LIN {X 0,Y 573.25,Z 574.073,A -85,B 0,C 180,E1 -2307.355,E2 -2307.355} C_VEL
LIN {X 0,Y 573.251,Z 574.074,A -85,B 0,C 180,E1 -2309.824,E2 -2309.824} C_VEL
LIN {X 0,Y 573.282,Z 574.075,A -85,B 0,C 180,E1 -2312.235,E2 -2312.235} C_VEL
LIN {X 0,Y 573.263,Z 574.072,A -85,B 0,C 180,E1 -2315.12,E2 -2315.12} C_VEL
LIN {X 0,Y 573.23,Z 574.076,A -85,B 0,C 180,E1 -2317.662,E2 -2317.662} C_VEL
LIN {X 0,Y 573.27,Z 574.075,A -85,B 0,C 180,E1 -2320.728,E2 -2320.728} C_VEL
LIN {X 0,Y 573.245,Z 574.074,A -85,B 0,C 180,E1 -2323.621,E2 -2323.621} C_VEL
LIN {X 0,Y 573.265,Z 574.072,A -85,B 0,C 180,E1 -2325.807,E2 -2325.807} C_VEL
LIN {X 0,Y 573.254,Z 574.076,A -85,B 0,C 180,E1 -2328.745,E2 -2328.745} C_VEL
LIN {X 0,Y 573.3,Z 574.067,A -85,B 0,C 180,E1 -2331.541,E2 -2331.541} C_VEL
LIN {X 0,Y 573.283,Z 574.078,A -85,B 0,C 180,E1 -2334.372,E2 -2334.372} C_VEL
LIN {X 0,Y 573.301,Z 574.07,A -85,B 0,C 180,E1 -2337.892,E2 -2337.892} C_VEL
LIN {X 0,Y 573.328,Z 574.067,A -85,B 0,C 180,E1 -2340.702,E2 -2340.702} C_VEL
LIN {X 0,Y 573.232,Z 574.076,A -85,B 0,C 180,E1 -2343.514,E2 -2343.514} C_VEL
LIN {X 0,Y 573.292,Z 574.069,A -85,B 0,C 180,E1 -2345.628,E2 -2345.628} C_VEL
LIN {X 0,Y 573.301,Z 574.074,A -85,B 0,C 180,E1 -2348.459,E2 -2348.459} C_VEL
LIN {X 0,Y 573.291,Z 574.068,A -85,B 0,C 180,E1 -2351.312,E2 -2351.312} C_VEL
LIN {X 0,Y 573.273,Z 574.08,A -85,B 0,C 180,E1 -2354.425,E2 -2354.425} C_VEL
LIN {X 0,Y 573.304,Z 574.233,A -85,B 0,C 180,E1 -2357.432,E2 -2357.432} C_VEL
LIN {X 0,Y 573.275,Z 587.865,A -85,B 0,C 180,E1 -2360.076,E2 -2360.076} C_VEL
LIN {X 0,Y 573.251,Z 593.888,A -85,B 0,C 180,E1 -2361.233,E2 -2361.233} C_VEL
LIN {X 0,Y 574.072,Z 600.547,A -85,B 0,C 180,E1 -2361.34,E2 -2361.34} C_VEL
LIN {X 0,Y 574.064,Z 601.305,A -85,B 0,C 180,E1 -2361.349,E2 -2361.349} C_VEL
LIN {X 0,Y 573.377,Z 607.149,A -85,B 0,C 180,E1 -2361.406,E2 -2361.406} C_VEL
LIN {X 0,Y 567.79,Z 626.154,A -85,B 0,C 180,E1 -2361.512,E2 -2361.512} C_VEL
LIN {X 0,Y 567.122,Z 631.997,A -85,B 0,C 180,E1 -2361.57,E2 -2361.57} C_VEL
LIN {X 0,Y 566.935,Z 700.341,A -85,B 0,C 180,E1 -2362.455,E2 -2362.455} C_VEL
LIN {X 0,Y 566.844,Z 713.428,A -85,B 0,C 180,E1 -2362.772,E2 -2362.772} C_VEL
LIN {X 0,Y 566.759,Z 725.192,A -85,B 0,C 180,E1 -2363.185,E2 -2363.185} C_VEL
LIN {X 0,Y 566.603,Z 736.809,A -85,B 0,C 180,E1 -2363.735,E2 -2363.735} C_VEL
LIN {X 0,Y 566.457,Z 748.669,A -85,B 0,C 180,E1 -2364.461,E2 -2364.461} C_VEL
LIN {X 0,Y 566.329,Z 758.973,A -85,B 0,C 180,E1 -2365.256,E2 -2365.256} C_VEL
LIN {X 0,Y 566.211,Z 768.35,A -85,B 0,C 180,E1 -2366.145,E2 -2366.145} C_VEL
LIN {X 0,Y 566.092,Z 777.03,A -85,B 0,C 180,E1 -2367.154,E2 -2367.154} C_VEL
LIN {X 0,Y 566.019,Z 785.144,A -85,B 0,C 180,E1 -2368.335,E2 -2368.335} C_VEL
LIN {X 0,Y 565.978,Z 790.458,A -85,B 0,C 180,E1 -2369.298,E2 -2369.298} C_VEL
LIN {X 0,Y 565.921,Z 796.115,A -85,B 0,C 180,E1 -2370.608,E2 -2370.608} C_VEL
LIN {X 0,Y 565.867,Z 799.979,A -85,B 0,C 180,E1 -2371.86,E2 -2371.86} C_VEL
LIN {X 0,Y 565.839,Z 802.539,A -85,B 0,C 180,E1 -2373.127,E2 -2373.127} C_VEL
LIN {X 0,Y 565.858,Z 803.553,A -85,B 0,C 180,E1 -2373.98,E2 -2373.98} C_VEL
LIN {X 0,Y 565.846,Z 803.984,A -85,B 0,C 180,E1 -2374.943,E2 -2374.943} C_VEL
LIN {X 0,Y 565.821,Z 803.511,A -85,B 0,C 180,E1 -2376.163,E2 -2376.163} C_VEL
LIN {X 0,Y 565.843,Z 801.631,A -85,B 0,C 180,E1 -2377.488,E2 -2377.488} C_VEL
LIN {X 0,Y 565.868,Z 799.217,A -85,B 0,C 180,E1 -2378.516,E2 -2378.516} C_VEL
LIN {X 0,Y 565.92,Z 795.465,A -85,B 0,C 180,E1 -2379.651,E2 -2379.651} C_VEL
LIN {X 0,Y 565.941,Z 789.748,A -85,B 0,C 180,E1 -2380.933,E2 -2380.933} C_VEL
LIN {X 0,Y 566.008,Z 782.933,A -85,B 0,C 180,E1 -2382.106,E2 -2382.106} C_VEL
LIN {X 0,Y 566.108,Z 776.028,A -85,B 0,C 180,E1 -2383.063,E2 -2383.063} C_VEL
LIN {X 0,Y 566.186,Z 767.481,A -85,B 0,C 180,E1 -2384.037,E2 -2384.037} C_VEL
LIN {X 0,Y 566.366,Z 757.173,A -85,B 0,C 180,E1 -2384.985,E2 -2384.985} C_VEL
LIN {X 0,Y 566.477,Z 746.803,A -85,B 0,C 180,E1 -2385.755,E2 -2385.755} C_VEL
LIN {X 0,Y 566.635,Z 735.245,A -85,B 0,C 180,E1 -2386.437,E2 -2386.437} C_VEL
LIN {X 0,Y 566.756,Z 722.817,A -85,B 0,C 180,E1 -2387,E2 -2387} C_VEL
LIN {X 0,Y 566.89,Z 709.938,A -85,B 0,C 180,E1 -2387.421,E2 -2387.421} C_VEL
LIN {X 0,Y 566.982,Z 696.718,A -85,B 0,C 180,E1 -2387.693,E2 -2387.693} C_VEL
LIN {X 0,Y 567.083,Z 599.04,A -85,B 0,C 180,E1 -2388.942,E2 -2388.942} C_VEL
LIN {X 0,Y 566.197,Z 593.841,A -85,B 0,C 180,E1 -2389.042,E2 -2389.042} C_VEL
LIN {X 0,Y 566.362,Z 579.311,A -85,B 0,C 180,E1 -2391.879,E2 -2391.879} C_VEL
LIN {X 0,Y 566.259,Z 574.948,A -85,B 0,C 180,E1 -2392.788,E2 -2392.788} C_VEL
LIN {X 0,Y 566.22,Z 574.957,A -85,B 0,C 180,E1 -2396.046,E2 -2396.046} C_VEL
LIN {X 0,Y 566.191,Z 574.953,A -85,B 0,C 180,E1 -2398.579,E2 -2398.579} C_VEL
LIN {X 0,Y 566.191,Z 574.951,A -85,B 0,C 180,E1 -2401.048,E2 -2401.048} C_VEL
LIN {X 0,Y 566.214,Z 574.95,A -85,B 0,C 180,E1 -2403.46,E2 -2403.46} C_VEL
LIN {X 0,Y 566.198,Z 574.956,A -85,B 0,C 180,E1 -2405.82,E2 -2405.82} C_VEL
LIN {X 0,Y 566.208,Z 574.95,A -85,B 0,C 180,E1 -2408.903,E2 -2408.903} C_VEL
LIN {X 0,Y 566.208,Z 574.949,A -85,B 0,C 180,E1 -2411.173,E2 -2411.173} C_VEL
LIN {X 0,Y 566.217,Z 574.948,A -85,B 0,C 180,E1 -2413.413,E2 -2413.413} C_VEL
LIN {X 0,Y 566.201,Z 574.96,A -85,B 0,C 180,E1 -2416.36,E2 -2416.36} C_VEL
LIN {X 0,Y 566.235,Z 574.951,A -85,B 0,C 180,E1 -2418.676,E2 -2418.676} C_VEL
LIN {X 0,Y 566.23,Z 574.947,A -85,B 0,C 180,E1 -2421.435,E2 -2421.435} C_VEL
LIN {X 0,Y 566.26,Z 574.951,A -85,B 0,C 180,E1 -2424.303,E2 -2424.303} C_VEL
LIN {X 0,Y 566.284,Z 574.941,A -85,B 0,C 180,E1 -2427.867,E2 -2427.867} C_VEL
LIN {X 0,Y 566.304,Z 574.945,A -85,B 0,C 180,E1 -2430.712,E2 -2430.712} C_VEL
LIN {X 0,Y 566.278,Z 574.947,A -85,B 0,C 180,E1 -2432.846,E2 -2432.846} C_VEL
LIN {X 0,Y 566.26,Z 574.943,A -85,B 0,C 180,E1 -2435.699,E2 -2435.699} C_VEL
LIN {X 0,Y 566.237,Z 574.954,A -85,B 0,C 180,E1 -2438.566,E2 -2438.566} C_VEL
LIN {X 0,Y 566.246,Z 574.945,A -85,B 0,C 180,E1 -2441.455,E2 -2441.455} C_VEL
LIN {X 0,Y 566.238,Z 574.951,A -85,B 0,C 180,E1 -2444.507,E2 -2444.507} C_VEL
LIN {X 0,Y 566.204,Z 574.953,A -85,B 0,C 180,E1 -2447.332,E2 -2447.332} C_VEL
LIN {X 0,Y 566.212,Z 574.951,A -85,B 0,C 180,E1 -2450.338,E2 -2450.338} C_VEL
LIN {X 0,Y 566.173,Z 574.959,A -85,B 0,C 180,E1 -2453.281,E2 -2453.281} C_VEL
LIN {X 0,Y 566.218,Z 574.949,A -85,B 0,C 180,E1 -2455.749,E2 -2455.749} C_VEL
LIN {X 0,Y 566.207,Z 574.95,A -85,B 0,C 180,E1 -2458.203,E2 -2458.203} C_VEL
LIN {X 0,Y 566.195,Z 574.961,A -85,B 0,C 180,E1 -2461.077,E2 -2461.077} C_VEL
LIN {X 0,Y 566.216,Z 574.95,A -85,B 0,C 180,E1 -2463.735,E2 -2463.735} C_VEL
LIN {X 0,Y 566.204,Z 574.951,A -85,B 0,C 180,E1 -2466.57,E2 -2466.57} C_VEL
LIN {X 0,Y 566.226,Z 574.951,A -85,B 0,C 180,E1 -2469.687,E2 -2469.687} C_VEL
LIN {X 0,Y 566.205,Z 574.953,A -85,B 0,C 180,E1 -2472.918,E2 -2472.918} C_VEL
LIN {X 0,Y 566.202,Z 574.951,A -85,B 0,C 180,E1 -2476.049,E2 -2476.049} C_VEL
LIN {X 0,Y 566.184,Z 574.954,A -85,B 0,C 180,E1 -2478.861,E2 -2478.861} C_VEL
LIN {X 0,Y 566.192,Z 574.959,A -85,B 0,C 180,E1 -2481.637,E2 -2481.637} C_VEL
LIN {X 0,Y 566.167,Z 574.955,A -85,B 0,C 180,E1 -2484.308,E2 -2484.308} C_VEL
LIN {X 0,Y 566.225,Z 574.948,A -85,B 0,C 180,E1 -2486.898,E2 -2486.898} C_VEL
LIN {X 0,Y 566.185,Z 574.959,A -85,B 0,C 180,E1 -2489.408,E2 -2489.408} C_VEL
LIN {X 0,Y 566.216,Z 574.956,A -85,B 0,C 180,E1 -2491.858,E2 -2491.858} C_VEL
LIN {X 0,Y 566.218,Z 574.95,A -85,B 0,C 180,E1 -2494.251,E2 -2494.251} C_VEL
LIN {X 0,Y 566.174,Z 574.953,A -85,B 0,C 180,E1 -2496.719,E2 -2496.719} C_VEL
LIN {X 0,Y 566.213,Z 574.956,A -85,B 0,C 180,E1 -2499.663,E2 -2499.663} C_VEL
LIN {X 0,Y 566.204,Z 574.95,A -85,B 0,C 180,E1 -2502.669,E2 -2502.669} C_VEL
LIN {X 0,Y 566.239,Z 574.951,A -85,B 0,C 180,E1 -2505.627,E2 -2505.627} C_VEL
LIN {X 0,Y 566.24,Z 574.946,A -85,B 0,C 180,E1 -2508.675,E2 -2508.675} C_VEL
LIN {X 0,Y 566.232,Z 574.948,A -85,B 0,C 180,E1 -2511.434,E2 -2511.434} C_VEL
LIN {X 0,Y 566.261,Z 574.949,A -85,B 0,C 180,E1 -2514.302,E2 -2514.302} C_VEL
LIN {X 0,Y 566.286,Z 574.945,A -85,B 0,C 180,E1 -2517.866,E2 -2517.866} C_VEL
LIN {X 0,Y 566.306,Z 574.94,A -85,B 0,C 180,E1 -2520.711,E2 -2520.711} C_VEL
LIN {X 0,Y 566.278,Z 574.942,A -85,B 0,C 180,E1 -2522.846,E2 -2522.846} C_VEL
LIN {X 0,Y 566.258,Z 574.945,A -85,B 0,C 180,E1 -2525.698,E2 -2525.698} C_VEL
LIN {X 0,Y 566.233,Z 574.953,A -85,B 0,C 180,E1 -2528.566,E2 -2528.566} C_VEL
LIN {X 0,Y 566.247,Z 574.944,A -85,B 0,C 180,E1 -2531.454,E2 -2531.454} C_VEL
LIN {X 0,Y 566.24,Z 574.955,A -85,B 0,C 180,E1 -2534.506,E2 -2534.506} C_VEL
LIN {X 0,Y 566.204,Z 574.95,A -85,B 0,C 180,E1 -2537.332,E2 -2537.332} C_VEL
LIN {X 0,Y 566.214,Z 574.955,A -85,B 0,C 180,E1 -2540.337,E2 -2540.337} C_VEL
LIN {X 0,Y 566.175,Z 574.955,A -85,B 0,C 180,E1 -2543.281,E2 -2543.281} C_VEL
LIN {X 0,Y 566.215,Z 574.948,A -85,B 0,C 180,E1 -2545.749,E2 -2545.749} C_VEL
LIN {X 0,Y 566.208,Z 574.952,A -85,B 0,C 180,E1 -2548.202,E2 -2548.202} C_VEL
LIN {X 0,Y 566.195,Z 574.956,A -85,B 0,C 180,E1 -2551.076,E2 -2551.076} C_VEL
LIN {X 0,Y 566.218,Z 574.948,A -85,B 0,C 180,E1 -2553.734,E2 -2553.734} C_VEL
LIN {X 0,Y 566.205,Z 574.955,A -85,B 0,C 180,E1 -2556.57,E2 -2556.57} C_VEL
LIN {X 0,Y 566.221,Z 574.948,A -85,B 0,C 180,E1 -2559.686,E2 -2559.686} C_VEL
LIN {X 0,Y 566.217,Z 574.948,A -85,B 0,C 180,E1 -2562.087,E2 -2562.087} C_VEL
LIN {X 0,Y 566.174,Z 574.964,A -85,B 0,C 180,E1 -2565.036,E2 -2565.036} C_VEL
LIN {X 0,Y 566.194,Z 574.951,A -85,B 0,C 180,E1 -2567.91,E2 -2567.91} C_VEL
LIN {X 0,Y 566.225,Z 574.951,A -85,B 0,C 180,E1 -2570.727,E2 -2570.727} C_VEL
LIN {X 0,Y 566.19,Z 574.953,A -85,B 0,C 180,E1 -2573.788,E2 -2573.788} C_VEL
LIN {X 0,Y 566.218,Z 574.949,A -85,B 0,C 180,E1 -2576.265,E2 -2576.265} C_VEL
LIN {X 0,Y 566.193,Z 574.956,A -85,B 0,C 180,E1 -2578.924,E2 -2578.924} C_VEL
LIN {X 0,Y 566.217,Z 574.952,A -85,B 0,C 180,E1 -2581.857,E2 -2581.857} C_VEL
LIN {X 0,Y 566.215,Z 574.952,A -85,B 0,C 180,E1 -2584.25,E2 -2584.25} C_VEL
LIN {X 0,Y 566.26,Z 575.009,A -85,B 0,C 180,E1 -2585.431,E2 -2585.431} C_VEL
LIN {X 0,Y 567.273,Z 580.215,A -85,B 0,C 180,E1 -2586.22,E2 -2586.22} C_VEL
LIN {X 0,Y 567.133,Z 596.227,A -85,B 0,C 180,E1 -2588.47,E2 -2588.47} C_VEL
LIN {X 0,Y 566.794,Z 618.681,A -85,B 0,C 180,E1 -2591.567,E2 -2591.567} C_VEL
LIN {X 0,Y 566.549,Z 637.787,A -85,B 0,C 180,E1 -2594.162,E2 -2594.162} C_VEL
LIN {X 0,Y 566.428,Z 651.349,A -85,B 0,C 180,E1 -2595.986,E2 -2595.986} C_VEL
LIN {X 0,Y 567.183,Z 658.149,A -85,B 0,C 180,E1 -2596.094,E2 -2596.094} C_VEL
LIN {X 0,Y 566.989,Z 759.91,A -85,B 0,C 180,E1 -2597.403,E2 -2597.403} C_VEL
LIN {X 0,Y 566.841,Z 772.433,A -85,B 0,C 180,E1 -2597.695,E2 -2597.695} C_VEL
LIN {X 0,Y 566.764,Z 785.356,A -85,B 0,C 180,E1 -2598.148,E2 -2598.148} C_VEL
LIN {X 0,Y 566.629,Z 797.14,A -85,B 0,C 180,E1 -2598.707,E2 -2598.707} C_VEL
LIN {X 0,Y 566.449,Z 809.192,A -85,B 0,C 180,E1 -2599.454,E2 -2599.454} C_VEL
LIN {X 0,Y 566.319,Z 819.592,A -85,B 0,C 180,E1 -2600.265,E2 -2600.265} C_VEL
LIN {X 0,Y 566.207,Z 828.105,A -85,B 0,C 180,E1 -2601.073,E2 -2601.073} C_VEL
LIN {X 0,Y 566.113,Z 835.955,A -85,B 0,C 180,E1 -2601.971,E2 -2601.971} C_VEL
LIN {X 0,Y 566.004,Z 843.617,A -85,B 0,C 180,E1 -2603.046,E2 -2603.046} C_VEL
LIN {X 0,Y 566.004,Z 850.676,A -85,B 0,C 180,E1 -2604.298,E2 -2604.298} C_VEL
LIN {X 0,Y 565.934,Z 855.369,A -85,B 0,C 180,E1 -2605.369,E2 -2605.369} C_VEL
LIN {X 0,Y 565.927,Z 858.955,A -85,B 0,C 180,E1 -2606.439,E2 -2606.439} C_VEL
LIN {X 0,Y 565.878,Z 860.806,A -85,B 0,C 180,E1 -2607.152,E2 -2607.152} C_VEL
LIN {X 0,Y 565.846,Z 863.185,A -85,B 0,C 180,E1 -2608.576,E2 -2608.576} C_VEL
LIN {X 0,Y 565.839,Z 864,A -85,B 0,C 180,E1 -2609.999,E2 -2609.999} C_VEL
LIN {X 0,Y 565.846,Z 863.187,A -85,B 0,C 180,E1 -2611.423,E2 -2611.423} C_VEL
LIN {X 0,Y 565.878,Z 860.812,A -85,B 0,C 180,E1 -2612.847,E2 -2612.847} C_VEL
LIN {X 0,Y 565.926,Z 857.898,A -85,B 0,C 180,E1 -2613.916,E2 -2613.916} C_VEL
LIN {X 0,Y 565.878,Z 853.952,A -85,B 0,C 180,E1 -2614.987,E2 -2614.987} C_VEL
LIN {X 0,Y 566.001,Z 848.871,A -85,B 0,C 180,E1 -2616.058,E2 -2616.058} C_VEL
LIN {X 0,Y 566.04,Z 842.474,A -85,B 0,C 180,E1 -2617.131,E2 -2617.131} C_VEL
LIN {X 0,Y 566.133,Z 834.485,A -85,B 0,C 180,E1 -2618.207,E2 -2618.207} C_VEL
LIN {X 0,Y 566.228,Z 826.344,A -85,B 0,C 180,E1 -2619.105,E2 -2619.105} C_VEL
LIN {X 0,Y 566.342,Z 816.411,A -85,B 0,C 180,E1 -2620.004,E2 -2620.004} C_VEL
LIN {X 0,Y 566.524,Z 805.296,A -85,B 0,C 180,E1 -2620.807,E2 -2620.807} C_VEL
LIN {X 0,Y 566.659,Z 794.194,A -85,B 0,C 180,E1 -2621.445,E2 -2621.445} C_VEL
LIN {X 0,Y 566.75,Z 782.006,A -85,B 0,C 180,E1 -2621.987,E2 -2621.987} C_VEL
LIN {X 0,Y 566.887,Z 769.211,A -85,B 0,C 180,E1 -2622.393,E2 -2622.393} C_VEL
LIN {X 0,Y 566.981,Z 757.164,A -85,B 0,C 180,E1 -2622.641,E2 -2622.641} C_VEL
LIN {X 0,Y 567.032,Z 655.343,A -85,B 0,C 180,E1 -2623.945,E2 -2623.945} C_VEL
LIN {X 0,Y 566.444,Z 651.276,A -85,B 0,C 180,E1 -2624.023,E2 -2624.023} C_VEL
LIN {X 0,Y 566.692,Z 627.248,A -85,B 0,C 180,E1 -2627.265,E2 -2627.265} C_VEL
LIN {X 0,Y 566.952,Z 606.411,A -85,B 0,C 180,E1 -2630.119,E2 -2630.119} C_VEL
LIN {X 0,Y 567.307,Z 584.574,A -85,B 0,C 180,E1 -2633.161,E2 -2633.161} C_VEL
LIN {X 0,Y 567.077,Z 578.976,A -85,B 0,C 180,E1 -2633.965,E2 -2633.965} C_VEL
LIN {X 0,Y 566.233,Z 574.957,A -85,B 0,C 180,E1 -2634.593,E2 -2634.593} C_VEL
LIN {X 0,Y 566.211,Z 574.952,A -85,B 0,C 180,E1 -2637.338,E2 -2637.338} C_VEL
LIN {X 0,Y 566.2,Z 574.953,A -85,B 0,C 180,E1 -2639.768,E2 -2639.768} C_VEL
LIN {X 0,Y 566.203,Z 574.96,A -85,B 0,C 180,E1 -2642.429,E2 -2642.429} C_VEL
LIN {X 0,Y 566.211,Z 574.953,A -85,B 0,C 180,E1 -2644.993,E2 -2644.993} C_VEL
LIN {X 0,Y 566.193,Z 574.952,A -85,B 0,C 180,E1 -2647.46,E2 -2647.46} C_VEL
LIN {X 0,Y 566.224,Z 574.954,A -85,B 0,C 180,E1 -2650.196,E2 -2650.196} C_VEL
LIN {X 0,Y 566.197,Z 574.954,A -85,B 0,C 180,E1 -2653.053,E2 -2653.053} C_VEL
LIN {X 0,Y 566.198,Z 574.955,A -85,B 0,C 180,E1 -2656.047,E2 -2656.047} C_VEL
LIN {X 0,Y 566.208,Z 574.954,A -85,B 0,C 180,E1 -2658.863,E2 -2658.863} C_VEL
LIN {X 0,Y 566.187,Z 574.953,A -85,B 0,C 180,E1 -2661.637,E2 -2661.637} C_VEL
LIN {X 0,Y 566.207,Z 574.957,A -85,B 0,C 180,E1 -2664.311,E2 -2664.311} C_VEL
LIN {X 0,Y 566.223,Z 574.951,A -85,B 0,C 180,E1 -2666.898,E2 -2666.898} C_VEL
LIN {X 0,Y 566.188,Z 574.952,A -85,B 0,C 180,E1 -2669.407,E2 -2669.407} C_VEL
LIN {X 0,Y 566.222,Z 574.949,A -85,B 0,C 180,E1 -2671.858,E2 -2671.858} C_VEL
LIN {X 0,Y 566.221,Z 574.955,A -85,B 0,C 180,E1 -2674.251,E2 -2674.251} C_VEL
LIN {X 0,Y 566.185,Z 574.958,A -85,B 0,C 180,E1 -2676.713,E2 -2676.713} C_VEL
LIN {X 0,Y 566.207,Z 574.95,A -85,B 0,C 180,E1 -2679.662,E2 -2679.662} C_VEL
LIN {X 0,Y 566.196,Z 574.957,A -85,B 0,C 180,E1 -2682.668,E2 -2682.668} C_VEL
LIN {X 0,Y 566.226,Z 574.948,A -85,B 0,C 180,E1 -2685.626,E2 -2685.626} C_VEL
LIN {X 0,Y 566.226,Z 574.953,A -85,B 0,C 180,E1 -2688.675,E2 -2688.675} C_VEL
LIN {X 0,Y 566.241,Z 574.946,A -85,B 0,C 180,E1 -2691.434,E2 -2691.434} C_VEL
LIN {X 0,Y 566.252,Z 574.955,A -85,B 0,C 180,E1 -2694.302,E2 -2694.302} C_VEL
LIN {X 0,Y 566.272,Z 574.945,A -85,B 0,C 180,E1 -2697.866,E2 -2697.866} C_VEL
LIN {X 0,Y 566.298,Z 574.943,A -85,B 0,C 180,E1 -2700.711,E2 -2700.711} C_VEL
LIN {X 0,Y 566.272,Z 574.945,A -85,B 0,C 180,E1 -2702.845,E2 -2702.845} C_VEL
LIN {X 0,Y 566.26,Z 574.946,A -85,B 0,C 180,E1 -2705.698,E2 -2705.698} C_VEL
LIN {X 0,Y 566.242,Z 574.952,A -85,B 0,C 180,E1 -2708.565,E2 -2708.565} C_VEL
LIN {X 0,Y 566.243,Z 574.946,A -85,B 0,C 180,E1 -2711.454,E2 -2711.454} C_VEL
LIN {X 0,Y 566.226,Z 574.957,A -85,B 0,C 180,E1 -2714.507,E2 -2714.507} C_VEL
LIN {X 0,Y 566.271,Z 575.092,A -85,B 0,C 180,E1 -2717.376,E2 -2717.376} C_VEL
LIN {X 0,Y 566.241,Z 588.233,A -85,B 0,C 180,E1 -2719.957,E2 -2719.957} C_VEL
LIN {X 0,Y 566.19,Z 593.854,A -85,B 0,C 180,E1 -2721.051,E2 -2721.051} C_VEL
LIN {X 0,Y 567.187,Z 600.576,A -85,B 0,C 180,E1 -2721.17,E2 -2721.17} C_VEL
LIN {X 0,Y 567.122,Z 631.997,A -85,B 0,C 180,E1 -2721.57,E2 -2721.57} C_VEL
LIN {X 0,Y 566.416,Z 635.921,A -85,B 0,C 180,E1 -2721.603,E2 -2721.603} C_VEL
LIN {X 0,Y 560.748,Z 648.204,A -85,B 0,C 180,E1 -2721.623,E2 -2721.623} C_VEL
LIN {X 0,Y 560.188,Z 652.117,A -85,B 0,C 180,E1 -2721.66,E2 -2721.66} C_VEL
LIN {X 0,Y 560.024,Z 700.973,A -85,B 0,C 180,E1 -2722.31,E2 -2722.31} C_VEL
LIN {X 0,Y 559.912,Z 713.82,A -85,B 0,C 180,E1 -2722.631,E2 -2722.631} C_VEL
LIN {X 0,Y 559.798,Z 725.266,A -85,B 0,C 180,E1 -2723.039,E2 -2723.039} C_VEL
LIN {X 0,Y 559.612,Z 737.425,A -85,B 0,C 180,E1 -2723.626,E2 -2723.626} C_VEL
LIN {X 0,Y 559.457,Z 748.173,A -85,B 0,C 180,E1 -2724.293,E2 -2724.293} C_VEL
LIN {X 0,Y 559.327,Z 758.049,A -85,B 0,C 180,E1 -2725.052,E2 -2725.052} C_VEL
LIN {X 0,Y 559.187,Z 767.063,A -85,B 0,C 180,E1 -2725.896,E2 -2725.896} C_VEL
LIN {X 0,Y 559.023,Z 775.909,A -85,B 0,C 180,E1 -2726.91,E2 -2726.91} C_VEL
LIN {X 0,Y 558.964,Z 783.819,A -85,B 0,C 180,E1 -2728.033,E2 -2728.033} C_VEL
LIN {X 0,Y 558.896,Z 790.145,A -85,B 0,C 180,E1 -2729.161,E2 -2729.161} C_VEL
LIN {X 0,Y 558.827,Z 794.778,A -85,B 0,C 180,E1 -2730.202,E2 -2730.202} C_VEL
LIN {X 0,Y 558.827,Z 798.325,A -85,B 0,C 180,E1 -2731.221,E2 -2731.221} C_VEL
LIN {X 0,Y 558.758,Z 801.643,A -85,B 0,C 180,E1 -2732.574,E2 -2732.574} C_VEL
LIN {X 0,Y 558.764,Z 803.491,A -85,B 0,C 180,E1 -2733.89,E2 -2733.89} C_VEL
LIN {X 0,Y 558.752,Z 803.981,A -85,B 0,C 180,E1 -2735.159,E2 -2735.159} C_VEL
LIN {X 0,Y 558.732,Z 803.288,A -85,B 0,C 180,E1 -2736.389,E2 -2736.389} C_VEL
LIN {X 0,Y 558.755,Z 801.489,A -85,B 0,C 180,E1 -2737.59,E2 -2737.59} C_VEL
LIN {X 0,Y 558.807,Z 798.043,A -85,B 0,C 180,E1 -2738.964,E2 -2738.964} C_VEL
LIN {X 0,Y 558.854,Z 792.793,A -85,B 0,C 180,E1 -2740.364,E2 -2740.364} C_VEL
LIN {X 0,Y 558.896,Z 786.646,A -85,B 0,C 180,E1 -2741.586,E2 -2741.586} C_VEL
LIN {X 0,Y 558.981,Z 779.074,A -85,B 0,C 180,E1 -2742.76,E2 -2742.76} C_VEL
LIN {X 0,Y 559.12,Z 770.156,A -85,B 0,C 180,E1 -2743.864,E2 -2743.864} C_VEL
LIN {X 0,Y 559.301,Z 760.04,A -85,B 0,C 180,E1 -2744.864,E2 -2744.864} C_VEL
LIN {X 0,Y 559.452,Z 749.138,A -85,B 0,C 180,E1 -2745.729,E2 -2745.729} C_VEL
LIN {X 0,Y 559.629,Z 738.117,A -85,B 0,C 180,E1 -2746.424,E2 -2746.424} C_VEL
LIN {X 0,Y 559.79,Z 727.068,A -85,B 0,C 180,E1 -2746.974,E2 -2746.974} C_VEL
LIN {X 0,Y 559.918,Z 714.065,A -85,B 0,C 180,E1 -2747.456,E2 -2747.456} C_VEL
LIN {X 0,Y 559.992,Z 701.471,A -85,B 0,C 180,E1 -2747.771,E2 -2747.771} C_VEL
LIN {X 0,Y 560.115,Z 670.961,A -85,B 0,C 180,E1 -2748.189,E2 -2748.189} C_VEL
LIN {X 0,Y 560.13,Z 599.387,A -85,B 0,C 180,E1 -2749.113,E2 -2749.113} C_VEL
LIN {X 0,Y 559.168,Z 593.853,A -85,B 0,C 180,E1 -2749.219,E2 -2749.219} C_VEL
LIN {X 0,Y 559.363,Z 578.134,A -85,B 0,C 180,E1 -2752.331,E2 -2752.331} C_VEL
LIN {X 0,Y 559.233,Z 575.824,A -85,B 0,C 180,E1 -2752.8,E2 -2752.8} C_VEL
LIN {X 0,Y 559.176,Z 575.834,A -85,B 0,C 180,E1 -2756.05,E2 -2756.05} C_VEL
LIN {X 0,Y 559.153,Z 575.828,A -85,B 0,C 180,E1 -2758.982,E2 -2758.982} C_VEL
LIN {X 0,Y 559.168,Z 575.83,A -85,B 0,C 180,E1 -2761.619,E2 -2761.619} C_VEL
LIN {X 0,Y 559.179,Z 575.832,A -85,B 0,C 180,E1 -2763.904,E2 -2763.904} C_VEL
LIN {X 0,Y 559.155,Z 575.831,A -85,B 0,C 180,E1 -2766.568,E2 -2766.568} C_VEL
LIN {X 0,Y 559.179,Z 575.825,A -85,B 0,C 180,E1 -2769.396,E2 -2769.396} C_VEL
LIN {X 0,Y 559.152,Z 575.831,A -85,B 0,C 180,E1 -2771.687,E2 -2771.687} C_VEL
LIN {X 0,Y 559.169,Z 575.831,A -85,B 0,C 180,E1 -2773.949,E2 -2773.949} C_VEL
LIN {X 0,Y 559.175,Z 575.834,A -85,B 0,C 180,E1 -2776.185,E2 -2776.185} C_VEL
LIN {X 0,Y 559.206,Z 575.827,A -85,B 0,C 180,E1 -2778.605,E2 -2778.605} C_VEL
LIN {X 0,Y 559.188,Z 575.824,A -85,B 0,C 180,E1 -2781.326,E2 -2781.326} C_VEL
LIN {X 0,Y 559.229,Z 575.825,A -85,B 0,C 180,E1 -2784.231,E2 -2784.231} C_VEL
LIN {X 0,Y 559.255,Z 575.817,A -85,B 0,C 180,E1 -2787.84,E2 -2787.84} C_VEL
LIN {X 0,Y 559.274,Z 575.821,A -85,B 0,C 180,E1 -2790.721,E2 -2790.721} C_VEL
LIN {X 0,Y 559.244,Z 575.822,A -85,B 0,C 180,E1 -2792.882,E2 -2792.882} C_VEL
LIN {X 0,Y 559.23,Z 575.819,A -85,B 0,C 180,E1 -2795.771,E2 -2795.771} C_VEL
LIN {X 0,Y 559.195,Z 575.833,A -85,B 0,C 180,E1 -2798.675,E2 -2798.675} C_VEL
LIN {X 0,Y 559.209,Z 575.821,A -85,B 0,C 180,E1 -2801.601,E2 -2801.601} C_VEL
LIN {X 0,Y 559.204,Z 575.828,A -85,B 0,C 180,E1 -2804.596,E2 -2804.596} C_VEL
LIN {X 0,Y 559.163,Z 575.828,A -85,B 0,C 180,E1 -2807.557,E2 -2807.557} C_VEL
LIN {X 0,Y 559.17,Z 575.826,A -85,B 0,C 180,E1 -2809.838,E2 -2809.838} C_VEL
LIN {X 0,Y 559.145,Z 575.83,A -85,B 0,C 180,E1 -2812.153,E2 -2812.153} C_VEL
LIN {X 0,Y 559.18,Z 575.83,A -85,B 0,C 180,E1 -2815.299,E2 -2815.299} C_VEL
LIN {X 0,Y 559.185,Z 575.825,A -85,B 0,C 180,E1 -2817.713,E2 -2817.713} C_VEL
LIN {X 0,Y 559.157,Z 575.828,A -85,B 0,C 180,E1 -2820.183,E2 -2820.183} C_VEL
LIN {X 0,Y 559.161,Z 575.831,A -85,B 0,C 180,E1 -2822.716,E2 -2822.716} C_VEL
LIN {X 0,Y 559.14,Z 575.838,A -85,B 0,C 180,E1 -2825.324,E2 -2825.324} C_VEL
LIN {X 0,Y 559.138,Z 575.83,A -85,B 0,C 180,E1 -2828.018,E2 -2828.018} C_VEL
LIN {X 0,Y 559.159,Z 575.83,A -85,B 0,C 180,E1 -2830.813,E2 -2830.813} C_VEL
LIN {X 0,Y 559.142,Z 575.833,A -85,B 0,C 180,E1 -2833.735,E2 -2833.735} C_VEL
LIN {X 0,Y 559.151,Z 575.83,A -85,B 0,C 180,E1 -2836.804,E2 -2836.804} C_VEL
LIN {X 0,Y 559.162,Z 575.833,A -85,B 0,C 180,E1 -2839.188,E2 -2839.188} C_VEL
LIN {X 0,Y 559.138,Z 575.833,A -85,B 0,C 180,E1 -2841.983,E2 -2841.983} C_VEL
LIN {X 0,Y 559.136,Z 575.831,A -85,B 0,C 180,E1 -2844.787,E2 -2844.787} C_VEL
LIN {X 0,Y 559.161,Z 575.834,A -85,B 0,C 180,E1 -2847.365,E2 -2847.365} C_VEL
LIN {X 0,Y 559.153,Z 575.831,A -85,B 0,C 180,E1 -2850.143,E2 -2850.143} C_VEL
LIN {X 0,Y 559.174,Z 575.827,A -85,B 0,C 180,E1 -2853.098,E2 -2853.098} C_VEL
LIN {X 0,Y 559.16,Z 575.833,A -85,B 0,C 180,E1 -2855.495,E2 -2855.495} C_VEL
LIN {X 0,Y 559.177,Z 575.825,A -85,B 0,C 180,E1 -2858.624,E2 -2858.624} C_VEL
LIN {X 0,Y 559.166,Z 575.826,A -85,B 0,C 180,E1 -2860.926,E2 -2860.926} C_VEL
LIN {X 0,Y 559.17,Z 575.836,A -85,B 0,C 180,E1 -2863.948,E2 -2863.948} C_VEL
LIN {X 0,Y 559.175,Z 575.832,A -85,B 0,C 180,E1 -2866.184,E2 -2866.184} C_VEL
LIN {X 0,Y 559.199,Z 575.823,A -85,B 0,C 180,E1 -2869.134,E2 -2869.134} C_VEL
LIN {X 0,Y 559.205,Z 575.832,A -85,B 0,C 180,E1 -2872.054,E2 -2872.054} C_VEL
LIN {X 0,Y 559.259,Z 575.815,A -85,B 0,C 180,E1 -2874.953,E2 -2874.953} C_VEL
LIN {X 0,Y 559.258,Z 575.82,A -85,B 0,C 180,E1 -2877.84,E2 -2877.84} C_VEL
LIN {X 0,Y 559.277,Z 575.815,A -85,B 0,C 180,E1 -2880.72,E2 -2880.72} C_VEL
LIN {X 0,Y 559.244,Z 575.818,A -85,B 0,C 180,E1 -2882.881,E2 -2882.881} C_VEL
LIN {X 0,Y 559.228,Z 575.821,A -85,B 0,C 180,E1 -2885.77,E2 -2885.77} C_VEL
LIN {X 0,Y 559.192,Z 575.828,A -85,B 0,C 180,E1 -2888.674,E2 -2888.674} C_VEL
LIN {X 0,Y 559.211,Z 575.821,A -85,B 0,C 180,E1 -2891.6,E2 -2891.6} C_VEL
LIN {X 0,Y 559.206,Z 575.83,A -85,B 0,C 180,E1 -2894.596,E2 -2894.596} C_VEL
LIN {X 0,Y 559.148,Z 575.829,A -85,B 0,C 180,E1 -2897.557,E2 -2897.557} C_VEL
LIN {X 0,Y 559.172,Z 575.827,A -85,B 0,C 180,E1 -2899.838,E2 -2899.838} C_VEL
LIN {X 0,Y 559.146,Z 575.832,A -85,B 0,C 180,E1 -2902.153,E2 -2902.153} C_VEL
LIN {X 0,Y 559.181,Z 575.826,A -85,B 0,C 180,E1 -2905.298,E2 -2905.298} C_VEL
LIN {X 0,Y 559.153,Z 575.828,A -85,B 0,C 180,E1 -2907.714,E2 -2907.714} C_VEL
LIN {X 0,Y 559.158,Z 575.83,A -85,B 0,C 180,E1 -2910.183,E2 -2910.183} C_VEL
LIN {X 0,Y 559.162,Z 575.836,A -85,B 0,C 180,E1 -2912.715,E2 -2912.715} C_VEL
LIN {X 0,Y 559.134,Z 575.833,A -85,B 0,C 180,E1 -2915.324,E2 -2915.324} C_VEL
LIN {X 0,Y 559.139,Z 575.83,A -85,B 0,C 180,E1 -2918.017,E2 -2918.017} C_VEL
LIN {X 0,Y 559.163,Z 575.835,A -85,B 0,C 180,E1 -2920.812,E2 -2920.812} C_VEL
LIN {X 0,Y 559.153,Z 575.835,A -85,B 0,C 180,E1 -2923.196,E2 -2923.196} C_VEL
LIN {X 0,Y 559.143,Z 575.83,A -85,B 0,C 180,E1 -2926.266,E2 -2926.266} C_VEL
LIN {X 0,Y 559.161,Z 575.836,A -85,B 0,C 180,E1 -2929.187,E2 -2929.187} C_VEL
LIN {X 0,Y 559.138,Z 575.83,A -85,B 0,C 180,E1 -2931.982,E2 -2931.982} C_VEL
LIN {X 0,Y 559.14,Z 575.834,A -85,B 0,C 180,E1 -2934.786,E2 -2934.786} C_VEL
LIN {X 0,Y 559.179,Z 575.834,A -85,B 0,C 180,E1 -2937.361,E2 -2937.361} C_VEL
LIN {X 0,Y 559.15,Z 575.83,A -85,B 0,C 180,E1 -2940.143,E2 -2940.143} C_VEL
LIN {X 0,Y 559.174,Z 575.834,A -85,B 0,C 180,E1 -2943.097,E2 -2943.097} C_VEL
LIN {X 0,Y 559.211,Z 575.841,A -85,B 0,C 180,E1 -2945.251,E2 -2945.251} C_VEL
LIN {X 0,Y 560.456,Z 583.194,A -85,B 0,C 180,E1 -2946.342,E2 -2946.342} C_VEL
LIN {X 0,Y 560.088,Z 603.669,A -85,B 0,C 180,E1 -2949.238,E2 -2949.238} C_VEL
LIN {X 0,Y 559.758,Z 625.505,A -85,B 0,C 180,E1 -2952.273,E2 -2952.273} C_VEL
LIN {X 0,Y 559.463,Z 646.221,A -85,B 0,C 180,E1 -2955.11,E2 -2955.11} C_VEL
LIN {X 0,Y 559.439,Z 651.349,A -85,B 0,C 180,E1 -2955.808,E2 -2955.808} C_VEL
LIN {X 0,Y 560.294,Z 658.175,A -85,B 0,C 180,E1 -2955.92,E2 -2955.92} C_VEL
LIN {X 0,Y 560.084,Z 759.91,A -85,B 0,C 180,E1 -2957.245,E2 -2957.245} C_VEL
LIN {X 0,Y 559.923,Z 772.433,A -85,B 0,C 180,E1 -2957.541,E2 -2957.541} C_VEL
LIN {X 0,Y 559.792,Z 785.358,A -85,B 0,C 180,E1 -2957.998,E2 -2957.998} C_VEL
LIN {X 0,Y 559.67,Z 796.795,A -85,B 0,C 180,E1 -2958.546,E2 -2958.546} C_VEL
LIN {X 0,Y 559.511,Z 807.899,A -85,B 0,C 180,E1 -2959.231,E2 -2959.231} C_VEL
LIN {X 0,Y 559.311,Z 818.532,A -85,B 0,C 180,E1 -2960.05,E2 -2960.05} C_VEL
LIN {X 0,Y 559.162,Z 828.106,A -85,B 0,C 180,E1 -2960.96,E2 -2960.96} C_VEL
LIN {X 0,Y 559.05,Z 835.955,A -85,B 0,C 180,E1 -2961.869,E2 -2961.869} C_VEL
LIN {X 0,Y 558.945,Z 843.617,A -85,B 0,C 180,E1 -2962.958,E2 -2962.958} C_VEL
LIN {X 0,Y 558.935,Z 850.676,A -85,B 0,C 180,E1 -2964.226,E2 -2964.226} C_VEL
LIN {X 0,Y 558.827,Z 855.369,A -85,B 0,C 180,E1 -2965.31,E2 -2965.31} C_VEL
LIN {X 0,Y 558.837,Z 858.955,A -85,B 0,C 180,E1 -2966.394,E2 -2966.394} C_VEL
LIN {X 0,Y 558.8,Z 860.806,A -85,B 0,C 180,E1 -2967.116,E2 -2967.116} C_VEL
LIN {X 0,Y 558.745,Z 863.184,A -85,B 0,C 180,E1 -2968.558,E2 -2968.558} C_VEL
LIN {X 0,Y 558.74,Z 864,A -85,B 0,C 180,E1 -2969.999,E2 -2969.999} C_VEL
LIN {X 0,Y 558.745,Z 863.187,A -85,B 0,C 180,E1 -2971.441,E2 -2971.441} C_VEL
LIN {X 0,Y 558.799,Z 860.812,A -85,B 0,C 180,E1 -2972.883,E2 -2972.883} C_VEL
LIN {X 0,Y 558.844,Z 857.898,A -85,B 0,C 180,E1 -2973.965,E2 -2973.965} C_VEL
LIN {X 0,Y 558.798,Z 853.952,A -85,B 0,C 180,E1 -2975.05,E2 -2975.05} C_VEL
LIN {X 0,Y 558.921,Z 848.871,A -85,B 0,C 180,E1 -2976.135,E2 -2976.135} C_VEL
LIN {X 0,Y 558.977,Z 842.474,A -85,B 0,C 180,E1 -2977.222,E2 -2977.222} C_VEL
LIN {X 0,Y 559.098,Z 834.485,A -85,B 0,C 180,E1 -2978.311,E2 -2978.311} C_VEL
LIN {X 0,Y 559.183,Z 826.344,A -85,B 0,C 180,E1 -2979.22,E2 -2979.22} C_VEL
LIN {X 0,Y 559.355,Z 816.411,A -85,B 0,C 180,E1 -2980.13,E2 -2980.13} C_VEL
LIN {X 0,Y 559.529,Z 805.376,A -85,B 0,C 180,E1 -2980.939,E2 -2980.939} C_VEL
LIN {X 0,Y 559.702,Z 793.16,A -85,B 0,C 180,E1 -2981.643,E2 -2981.643} C_VEL
LIN {X 0,Y 559.83,Z 780.792,A -85,B 0,C 180,E1 -2982.184,E2 -2982.184} C_VEL
LIN {X 0,Y 559.934,Z 767.382,A -85,B 0,C 180,E1 -2982.596,E2 -2982.596} C_VEL
LIN {X 0,Y 560.087,Z 754.146,A -85,B 0,C 180,E1 -2982.845,E2 -2982.845} C_VEL
LIN {X 0,Y 560.12,Z 655.762,A -85,B 0,C 180,E1 -2984.116,E2 -2984.116} C_VEL
LIN {X 0,Y 559.457,Z 651.276,A -85,B 0,C 180,E1 -2984.202,E2 -2984.202} C_VEL
LIN {X 0,Y 559.71,Z 628.861,A -85,B 0,C 180,E1 -2987.265,E2 -2987.265} C_VEL
LIN {X 0,Y 560.023,Z 607.775,A -85,B 0,C 180,E1 -2990.188,E2 -2990.188} C_VEL
LIN {X 0,Y 560.428,Z 585.939,A -85,B 0,C 180,E1 -2993.266,E2 -2993.266} C_VEL
LIN {X 0,Y 560.437,Z 581.953,A -85,B 0,C 180,E1 -2993.834,E2 -2993.834} C_VEL
LIN {X 0,Y 559.205,Z 575.832,A -85,B 0,C 180,E1 -2994.747,E2 -2994.747} C_VEL
LIN {X 0,Y 559.188,Z 575.827,A -85,B 0,C 180,E1 -2997.711,E2 -2997.711} C_VEL
LIN {X 0,Y 559.152,Z 575.834,A -85,B 0,C 180,E1 -3000.182,E2 -3000.182} C_VEL
LIN {X 0,Y 559.173,Z 575.835,A -85,B 0,C 180,E1 -3002.713,E2 -3002.713} C_VEL
LIN {X 0,Y 559.156,Z 575.83,A -85,B 0,C 180,E1 -3005.321,E2 -3005.321} C_VEL
LIN {X 0,Y 559.132,Z 575.835,A -85,B 0,C 180,E1 -3008.016,E2 -3008.016} C_VEL
LIN {X 0,Y 559.173,Z 575.833,A -85,B 0,C 180,E1 -3010.81,E2 -3010.81} C_VEL
LIN {X 0,Y 559.137,Z 575.833,A -85,B 0,C 180,E1 -3013.733,E2 -3013.733} C_VEL
LIN {X 0,Y 559.164,Z 575.833,A -85,B 0,C 180,E1 -3016.8,E2 -3016.8} C_VEL
LIN {X 0,Y 559.172,Z 575.828,A -85,B 0,C 180,E1 -3019.189,E2 -3019.189} C_VEL
LIN {X 0,Y 559.131,Z 575.834,A -85,B 0,C 180,E1 -3021.982,E2 -3021.982} C_VEL
LIN {X 0,Y 559.154,Z 575.833,A -85,B 0,C 180,E1 -3024.782,E2 -3024.782} C_VEL
LIN {X 0,Y 559.168,Z 575.827,A -85,B 0,C 180,E1 -3027.361,E2 -3027.361} C_VEL
LIN {X 0,Y 559.183,Z 575.83,A -85,B 0,C 180,E1 -3030.134,E2 -3030.134} C_VEL
LIN {X 0,Y 559.176,Z 575.826,A -85,B 0,C 180,E1 -3033.169,E2 -3033.169} C_VEL
LIN {X 0,Y 559.15,Z 575.829,A -85,B 0,C 180,E1 -3035.494,E2 -3035.494} C_VEL
LIN {X 0,Y 559.164,Z 575.833,A -85,B 0,C 180,E1 -3038.623,E2 -3038.623} C_VEL
LIN {X 0,Y 559.164,Z 575.83,A -85,B 0,C 180,E1 -3040.926,E2 -3040.926} C_VEL
LIN {X 0,Y 559.161,Z 575.831,A -85,B 0,C 180,E1 -3043.948,E2 -3043.948} C_VEL
LIN {X 0,Y 559.166,Z 575.834,A -85,B 0,C 180,E1 -3046.184,E2 -3046.184} C_VEL
LIN {X 0,Y 559.188,Z 575.825,A -85,B 0,C 180,E1 -3049.133,E2 -3049.133} C_VEL
LIN {X 0,Y 559.201,Z 575.828,A -85,B 0,C 180,E1 -3052.053,E2 -3052.053} C_VEL
LIN {X 0,Y 559.252,Z 575.818,A -85,B 0,C 180,E1 -3054.953,E2 -3054.953} C_VEL
LIN {X 0,Y 559.244,Z 575.821,A -85,B 0,C 180,E1 -3057.839,E2 -3057.839} C_VEL
LIN {X 0,Y 559.268,Z 575.819,A -85,B 0,C 180,E1 -3060.72,E2 -3060.72} C_VEL
LIN {X 0,Y 559.237,Z 575.821,A -85,B 0,C 180,E1 -3062.881,E2 -3062.881} C_VEL
LIN {X 0,Y 559.23,Z 575.823,A -85,B 0,C 180,E1 -3065.77,E2 -3065.77} C_VEL
LIN {X 0,Y 559.197,Z 575.828,A -85,B 0,C 180,E1 -3068.674,E2 -3068.674} C_VEL
LIN {X 0,Y 559.201,Z 575.825,A -85,B 0,C 180,E1 -3071.6,E2 -3071.6} C_VEL
LIN {X 0,Y 559.191,Z 575.832,A -85,B 0,C 180,E1 -3074.596,E2 -3074.596} C_VEL
LIN {X 0,Y 559.252,Z 575.917,A -85,B 0,C 180,E1 -3077.312,E2 -3077.312} C_VEL
LIN {X 0,Y 559.237,Z 587.012,A -85,B 0,C 180,E1 -3079.522,E2 -3079.522} C_VEL
LIN {X 0,Y 559.176,Z 593.843,A -85,B 0,C 180,E1 -3080.869,E2 -3080.869} C_VEL
LIN {X 0,Y 560.297,Z 600.391,A -85,B 0,C 180,E1 -3080.994,E2 -3080.994} C_VEL
LIN {X 0,Y 560.188,Z 652.117,A -85,B 0,C 180,E1 -3081.66,E2 -3081.66} C_VEL
LIN {X 0,Y 559.685,Z 657.956,A -85,B 0,C 180,E1 -3081.723,E2 -3081.723} C_VEL
LIN {X 0,Y 556.856,Z 667.442,A -85,B 0,C 180,E1 -3081.777,E2 -3081.777} C_VEL
LIN {X 0,Y 553.886,Z 676.93,A -85,B 0,C 180,E1 -3081.829,E2 -3081.829} C_VEL
LIN {X 0,Y 553.171,Z 682.783,A -85,B 0,C 180,E1 -3081.888,E2 -3081.888} C_VEL
LIN {X 0,Y 553.108,Z 702.341,A -85,B 0,C 180,E1 -3082.176,E2 -3082.176} C_VEL
LIN {X 0,Y 552.961,Z 714.256,A -85,B 0,C 180,E1 -3082.488,E2 -3082.488} C_VEL
LIN {X 0,Y 552.831,Z 725.927,A -85,B 0,C 180,E1 -3082.913,E2 -3082.913} C_VEL
LIN {X 0,Y 552.63,Z 737.79,A -85,B 0,C 180,E1 -3083.501,E2 -3083.501} C_VEL
LIN {X 0,Y 552.467,Z 749.099,A -85,B 0,C 180,E1 -3084.221,E2 -3084.221} C_VEL
LIN {X 0,Y 552.288,Z 758.85,A -85,B 0,C 180,E1 -3084.993,E2 -3084.993} C_VEL
LIN {X 0,Y 552.133,Z 767.708,A -85,B 0,C 180,E1 -3085.846,E2 -3085.846} C_VEL
LIN {X 0,Y 551.987,Z 777.185,A -85,B 0,C 180,E1 -3086.971,E2 -3086.971} C_VEL
LIN {X 0,Y 551.889,Z 784.839,A -85,B 0,C 180,E1 -3088.111,E2 -3088.111} C_VEL
LIN {X 0,Y 551.805,Z 791.475,A -85,B 0,C 180,E1 -3089.364,E2 -3089.364} C_VEL
LIN {X 0,Y 551.734,Z 796.587,A -85,B 0,C 180,E1 -3090.632,E2 -3090.632} C_VEL
LIN {X 0,Y 551.675,Z 800.313,A -85,B 0,C 180,E1 -3091.917,E2 -3091.917} C_VEL
LIN {X 0,Y 551.659,Z 802.745,A -85,B 0,C 180,E1 -3093.217,E2 -3093.217} C_VEL
LIN {X 0,Y 551.655,Z 803.646,A -85,B 0,C 180,E1 -3094.099,E2 -3094.099} C_VEL
LIN {X 0,Y 551.666,Z 803.934,A -85,B 0,C 180,E1 -3095.382,E2 -3095.382} C_VEL
LIN {X 0,Y 551.645,Z 802.876,A -85,B 0,C 180,E1 -3096.783,E2 -3096.783} C_VEL
LIN {X 0,Y 551.658,Z 801.041,A -85,B 0,C 180,E1 -3097.829,E2 -3097.829} C_VEL
LIN {X 0,Y 551.712,Z 798.057,A -85,B 0,C 180,E1 -3099.01,E2 -3099.01} C_VEL
LIN {X 0,Y 551.741,Z 793.955,A -85,B 0,C 180,E1 -3100.159,E2 -3100.159} C_VEL
LIN {X 0,Y 551.813,Z 787.722,A -85,B 0,C 180,E1 -3101.474,E2 -3101.474} C_VEL
LIN {X 0,Y 551.914,Z 780.245,A -85,B 0,C 180,E1 -3102.694,E2 -3102.694} C_VEL
LIN {X 0,Y 552.071,Z 771.661,A -85,B 0,C 180,E1 -3103.805,E2 -3103.805} C_VEL
LIN {X 0,Y 552.225,Z 762.941,A -85,B 0,C 180,E1 -3104.723,E2 -3104.723} C_VEL
LIN {X 0,Y 552.408,Z 752.765,A -85,B 0,C 180,E1 -3105.596,E2 -3105.596} C_VEL
LIN {X 0,Y 552.559,Z 741.894,A -85,B 0,C 180,E1 -3106.347,E2 -3106.347} C_VEL
LIN {X 0,Y 552.794,Z 730.515,A -85,B 0,C 180,E1 -3106.968,E2 -3106.968} C_VEL
LIN {X 0,Y 552.954,Z 717.768,A -85,B 0,C 180,E1 -3107.491,E2 -3107.491} C_VEL
LIN {X 0,Y 553.058,Z 704.466,A -85,B 0,C 180,E1 -3107.872,E2 -3107.872} C_VEL
LIN {X 0,Y 553.17,Z 689.133,A -85,B 0,C 180,E1 -3108.119,E2 -3108.119} C_VEL
LIN {X 0,Y 553.352,Z 600.793,A -85,B 0,C 180,E1 -3109.271,E2 -3109.271} C_VEL
LIN {X 0,Y 552.155,Z 593.845,A -85,B 0,C 180,E1 -3109.404,E2 -3109.404} C_VEL
LIN {X 0,Y 552.316,Z 578.001,A -85,B 0,C 180,E1 -3112.585,E2 -3112.585} C_VEL
LIN {X 0,Y 552.195,Z 576.701,A -85,B 0,C 180,E1 -3112.862,E2 -3112.862} C_VEL
LIN {X 0,Y 552.138,Z 576.712,A -85,B 0,C 180,E1 -3115.941,E2 -3115.941} C_VEL
LIN {X 0,Y 552.115,Z 576.707,A -85,B 0,C 180,E1 -3118.541,E2 -3118.541} C_VEL
LIN {X 0,Y 552.123,Z 576.706,A -85,B 0,C 180,E1 -3121.438,E2 -3121.438} C_VEL
LIN {X 0,Y 552.128,Z 576.709,A -85,B 0,C 180,E1 -3124.357,E2 -3124.357} C_VEL
LIN {X 0,Y 552.109,Z 576.707,A -85,B 0,C 180,E1 -3126.759,E2 -3126.759} C_VEL
LIN {X 0,Y 552.12,Z 576.704,A -85,B 0,C 180,E1 -3129.121,E2 -3129.121} C_VEL
LIN {X 0,Y 552.128,Z 576.704,A -85,B 0,C 180,E1 -3131.445,E2 -3131.445} C_VEL
LIN {X 0,Y 552.118,Z 576.707,A -85,B 0,C 180,E1 -3133.738,E2 -3133.738} C_VEL
LIN {X 0,Y 552.138,Z 576.708,A -85,B 0,C 180,E1 -3136.005,E2 -3136.005} C_VEL
LIN {X 0,Y 552.163,Z 576.7,A -85,B 0,C 180,E1 -3138.994,E2 -3138.994} C_VEL
LIN {X 0,Y 552.16,Z 576.703,A -85,B 0,C 180,E1 -3141.952,E2 -3141.952} C_VEL
LIN {X 0,Y 552.227,Z 576.694,A -85,B 0,C 180,E1 -3144.89,E2 -3144.89} C_VEL
LIN {X 0,Y 552.227,Z 576.692,A -85,B 0,C 180,E1 -3147.813,E2 -3147.813} C_VEL
LIN {X 0,Y 552.245,Z 576.696,A -85,B 0,C 180,E1 -3150.73,E2 -3150.73} C_VEL
LIN {X 0,Y 552.21,Z 576.698,A -85,B 0,C 180,E1 -3152.919,E2 -3152.919} C_VEL
LIN {X 0,Y 552.2,Z 576.695,A -85,B 0,C 180,E1 -3155.845,E2 -3155.845} C_VEL
LIN {X 0,Y 552.165,Z 576.708,A -85,B 0,C 180,E1 -3158.786,E2 -3158.786} C_VEL
LIN {X 0,Y 552.166,Z 576.698,A -85,B 0,C 180,E1 -3161.751,E2 -3161.751} C_VEL
LIN {X 0,Y 552.141,Z 576.711,A -85,B 0,C 180,E1 -3164.749,E2 -3164.749} C_VEL
LIN {X 0,Y 552.113,Z 576.705,A -85,B 0,C 180,E1 -3167.789,E2 -3167.789} C_VEL
LIN {X 0,Y 552.131,Z 576.703,A -85,B 0,C 180,E1 -3170.102,E2 -3170.102} C_VEL
LIN {X 0,Y 552.096,Z 576.71,A -85,B 0,C 180,E1 -3172.452,E2 -3172.452} C_VEL
LIN {X 0,Y 552.16,Z 576.704,A -85,B 0,C 180,E1 -3175.351,E2 -3175.351} C_VEL
LIN {X 0,Y 552.124,Z 576.704,A -85,B 0,C 180,E1 -3178.098,E2 -3178.098} C_VEL
LIN {X 0,Y 552.106,Z 576.709,A -85,B 0,C 180,E1 -3180.61,E2 -3180.61} C_VEL
LIN {X 0,Y 552.12,Z 576.714,A -85,B 0,C 180,E1 -3183.186,E2 -3183.186} C_VEL
LIN {X 0,Y 552.093,Z 576.709,A -85,B 0,C 180,E1 -3185.844,E2 -3185.844} C_VEL
LIN {X 0,Y 552.13,Z 576.71,A -85,B 0,C 180,E1 -3189.062,E2 -3189.062} C_VEL
LIN {X 0,Y 552.125,Z 576.712,A -85,B 0,C 180,E1 -3191.446,E2 -3191.446} C_VEL
LIN {X 0,Y 552.095,Z 576.708,A -85,B 0,C 180,E1 -3194.532,E2 -3194.532} C_VEL
LIN {X 0,Y 552.135,Z 576.71,A -85,B 0,C 180,E1 -3197.585,E2 -3197.585} C_VEL
LIN {X 0,Y 552.134,Z 576.702,A -85,B 0,C 180,E1 -3200.473,E2 -3200.473} C_VEL
LIN {X 0,Y 552.111,Z 576.712,A -85,B 0,C 180,E1 -3203.317,E2 -3203.317} C_VEL
LIN {X 0,Y 552.132,Z 576.707,A -85,B 0,C 180,E1 -3205.939,E2 -3205.939} C_VEL
LIN {X 0,Y 552.124,Z 576.704,A -85,B 0,C 180,E1 -3208.541,E2 -3208.541} C_VEL
LIN {X 0,Y 552.129,Z 576.709,A -85,B 0,C 180,E1 -3211.438,E2 -3211.438} C_VEL
LIN {X 0,Y 552.135,Z 576.704,A -85,B 0,C 180,E1 -3214.356,E2 -3214.356} C_VEL
LIN {X 0,Y 552.101,Z 576.707,A -85,B 0,C 180,E1 -3216.758,E2 -3216.758} C_VEL
LIN {X 0,Y 552.123,Z 576.705,A -85,B 0,C 180,E1 -3219.12,E2 -3219.12} C_VEL
LIN {X 0,Y 552.125,Z 576.707,A -85,B 0,C 180,E1 -3221.444,E2 -3221.444} C_VEL
LIN {X 0,Y 552.12,Z 576.712,A -85,B 0,C 180,E1 -3223.737,E2 -3223.737} C_VEL
LIN {X 0,Y 552.14,Z 576.711,A -85,B 0,C 180,E1 -3226.005,E2 -3226.005} C_VEL
LIN {X 0,Y 552.167,Z 576.698,A -85,B 0,C 180,E1 -3228.994,E2 -3228.994} C_VEL
LIN {X 0,Y 552.16,Z 576.708,A -85,B 0,C 180,E1 -3231.952,E2 -3231.952} C_VEL
LIN {X 0,Y 552.233,Z 576.691,A -85,B 0,C 180,E1 -3234.889,E2 -3234.889} C_VEL
LIN {X 0,Y 552.229,Z 576.695,A -85,B 0,C 180,E1 -3237.812,E2 -3237.812} C_VEL
LIN {X 0,Y 552.247,Z 576.691,A -85,B 0,C 180,E1 -3240.729,E2 -3240.729} C_VEL
LIN {X 0,Y 552.21,Z 576.694,A -85,B 0,C 180,E1 -3242.918,E2 -3242.918} C_VEL
LIN {X 0,Y 552.199,Z 576.698,A -85,B 0,C 180,E1 -3245.844,E2 -3245.844} C_VEL
LIN {X 0,Y 552.159,Z 576.703,A -85,B 0,C 180,E1 -3248.786,E2 -3248.786} C_VEL
LIN {X 0,Y 552.168,Z 576.7,A -85,B 0,C 180,E1 -3251.75,E2 -3251.75} C_VEL
LIN {X 0,Y 552.142,Z 576.707,A -85,B 0,C 180,E1 -3254.748,E2 -3254.748} C_VEL
LIN {X 0,Y 552.106,Z 576.707,A -85,B 0,C 180,E1 -3257.789,E2 -3257.789} C_VEL
LIN {X 0,Y 552.133,Z 576.706,A -85,B 0,C 180,E1 -3260.101,E2 -3260.101} C_VEL
LIN {X 0,Y 552.097,Z 576.715,A -85,B 0,C 180,E1 -3262.451,E2 -3262.451} C_VEL
LIN {X 0,Y 552.161,Z 576.7,A -85,B 0,C 180,E1 -3265.35,E2 -3265.35} C_VEL
LIN {X 0,Y 552.111,Z 576.707,A -85,B 0,C 180,E1 -3268.098,E2 -3268.098} C_VEL
LIN {X 0,Y 552.108,Z 576.714,A -85,B 0,C 180,E1 -3270.609,E2 -3270.609} C_VEL
LIN {X 0,Y 552.121,Z 576.708,A -85,B 0,C 180,E1 -3273.186,E2 -3273.186} C_VEL
LIN {X 0,Y 552.091,Z 576.708,A -85,B 0,C 180,E1 -3275.843,E2 -3275.843} C_VEL
LIN {X 0,Y 552.123,Z 576.709,A -85,B 0,C 180,E1 -3278.589,E2 -3278.589} C_VEL
LIN {X 0,Y 552.136,Z 576.705,A -85,B 0,C 180,E1 -3281.445,E2 -3281.445} C_VEL
LIN {X 0,Y 552.099,Z 576.71,A -85,B 0,C 180,E1 -3284.531,E2 -3284.531} C_VEL
LIN {X 0,Y 552.135,Z 576.705,A -85,B 0,C 180,E1 -3287.584,E2 -3287.584} C_VEL
LIN {X 0,Y 552.138,Z 576.703,A -85,B 0,C 180,E1 -3290.473,E2 -3290.473} C_VEL
LIN {X 0,Y 552.112,Z 576.713,A -85,B 0,C 180,E1 -3293.317,E2 -3293.317} C_VEL
LIN {X 0,Y 552.135,Z 576.704,A -85,B 0,C 180,E1 -3295.939,E2 -3295.939} C_VEL
LIN {X 0,Y 552.125,Z 576.705,A -85,B 0,C 180,E1 -3298.54,E2 -3298.54} C_VEL
LIN {X 0,Y 552.13,Z 576.713,A -85,B 0,C 180,E1 -3301.438,E2 -3301.438} C_VEL
LIN {X 0,Y 552.134,Z 576.707,A -85,B 0,C 180,E1 -3304.355,E2 -3304.355} C_VEL
LIN {X 0,Y 552.205,Z 576.749,A -85,B 0,C 180,E1 -3305.088,E2 -3305.088} C_VEL
LIN {X 0,Y 553.516,Z 584.242,A -85,B 0,C 180,E1 -3306.216,E2 -3306.216} C_VEL
LIN {X 0,Y 553.214,Z 602.304,A -85,B 0,C 180,E1 -3308.772,E2 -3308.772} C_VEL
LIN {X 0,Y 552.854,Z 622.775,A -85,B 0,C 180,E1 -3311.661,E2 -3311.661} C_VEL
LIN {X 0,Y 552.499,Z 643.246,A -85,B 0,C 180,E1 -3314.506,E2 -3314.506} C_VEL
LIN {X 0,Y 552.443,Z 651.349,A -85,B 0,C 180,E1 -3315.624,E2 -3315.624} C_VEL
LIN {X 0,Y 553.416,Z 659.242,A -85,B 0,C 180,E1 -3315.755,E2 -3315.755} C_VEL
LIN {X 0,Y 553.177,Z 759.91,A -85,B 0,C 180,E1 -3317.083,E2 -3317.083} C_VEL
LIN {X 0,Y 553.015,Z 772.432,A -85,B 0,C 180,E1 -3317.383,E2 -3317.383} C_VEL
LIN {X 0,Y 552.863,Z 785.351,A -85,B 0,C 180,E1 -3317.845,E2 -3317.845} C_VEL
LIN {X 0,Y 552.692,Z 797.651,A -85,B 0,C 180,E1 -3318.448,E2 -3318.448} C_VEL
LIN {X 0,Y 552.471,Z 809.188,A -85,B 0,C 180,E1 -3319.184,E2 -3319.184} C_VEL
LIN {X 0,Y 552.27,Z 819.594,A -85,B 0,C 180,E1 -3320.014,E2 -3320.014} C_VEL
LIN {X 0,Y 552.126,Z 828.106,A -85,B 0,C 180,E1 -3320.844,E2 -3320.844} C_VEL
LIN {X 0,Y 552.013,Z 835.955,A -85,B 0,C 180,E1 -3321.764,E2 -3321.764} C_VEL
LIN {X 0,Y 551.89,Z 843.616,A -85,B 0,C 180,E1 -3322.867,E2 -3322.867} C_VEL
LIN {X 0,Y 551.867,Z 850.676,A -85,B 0,C 180,E1 -3324.152,E2 -3324.152} C_VEL
LIN {X 0,Y 551.725,Z 855.369,A -85,B 0,C 180,E1 -3325.25,E2 -3325.25} C_VEL
LIN {X 0,Y 551.751,Z 858.956,A -85,B 0,C 180,E1 -3326.348,E2 -3326.348} C_VEL
LIN {X 0,Y 551.724,Z 860.806,A -85,B 0,C 180,E1 -3327.079,E2 -3327.079} C_VEL
LIN {X 0,Y 551.645,Z 863.184,A -85,B 0,C 180,E1 -3328.539,E2 -3328.539} C_VEL
LIN {X 0,Y 551.64,Z 864,A -85,B 0,C 180,E1 -3329.999,E2 -3329.999} C_VEL
LIN {X 0,Y 551.645,Z 863.186,A -85,B 0,C 180,E1 -3331.459,E2 -3331.459} C_VEL
LIN {X 0,Y 551.724,Z 860.812,A -85,B 0,C 180,E1 -3332.92,E2 -3332.92} C_VEL
LIN {X 0,Y 551.764,Z 857.898,A -85,B 0,C 180,E1 -3334.016,E2 -3334.016} C_VEL
LIN {X 0,Y 551.724,Z 853.952,A -85,B 0,C 180,E1 -3335.115,E2 -3335.115} C_VEL
LIN {X 0,Y 551.814,Z 848.128,A -85,B 0,C 180,E1 -3336.353,E2 -3336.353} C_VEL
LIN {X 0,Y 551.926,Z 841.242,A -85,B 0,C 180,E1 -3337.499,E2 -3337.499} C_VEL
LIN {X 0,Y 552.082,Z 832.998,A -85,B 0,C 180,E1 -3338.602,E2 -3338.602} C_VEL
LIN {X 0,Y 552.22,Z 824.548,A -85,B 0,C 180,E1 -3339.522,E2 -3339.522} C_VEL
LIN {X 0,Y 552.425,Z 814.107,A -85,B 0,C 180,E1 -3340.444,E2 -3340.444} C_VEL
LIN {X 0,Y 552.581,Z 803.144,A -85,B 0,C 180,E1 -3341.223,E2 -3341.223} C_VEL
LIN {X 0,Y 552.78,Z 792.425,A -85,B 0,C 180,E1 -3341.829,E2 -3341.829} C_VEL
LIN {X 0,Y 552.899,Z 780.788,A -85,B 0,C 180,E1 -3342.339,E2 -3342.339} C_VEL
LIN {X 0,Y 553.001,Z 767.381,A -85,B 0,C 180,E1 -3342.756,E2 -3342.756} C_VEL
LIN {X 0,Y 553.166,Z 754.146,A -85,B 0,C 180,E1 -3343.009,E2 -3343.009} C_VEL
LIN {X 0,Y 553.302,Z 656.93,A -85,B 0,C 180,E1 -3344.278,E2 -3344.278} C_VEL
LIN {X 0,Y 552.442,Z 651.276,A -85,B 0,C 180,E1 -3344.386,E2 -3344.386} C_VEL
LIN {X 0,Y 552.748,Z 629.574,A -85,B 0,C 180,E1 -3347.389,E2 -3347.389} C_VEL
LIN {X 0,Y 553.09,Z 609.14,A -85,B 0,C 180,E1 -3350.258,E2 -3350.258} C_VEL
LIN {X 0,Y 553.476,Z 588.415,A -85,B 0,C 180,E1 -3353.18,E2 -3353.18} C_VEL
LIN {X 0,Y 553.385,Z 582.771,A -85,B 0,C 180,E1 -3353.978,E2 -3353.978} C_VEL
LIN {X 0,Y 552.183,Z 576.706,A -85,B 0,C 180,E1 -3354.911,E2 -3354.911} C_VEL
LIN {X 0,Y 552.122,Z 576.71,A -85,B 0,C 180,E1 -3358.097,E2 -3358.097} C_VEL
LIN {X 0,Y 552.101,Z 576.718,A -85,B 0,C 180,E1 -3360.608,E2 -3360.608} C_VEL
LIN {X 0,Y 552.121,Z 576.707,A -85,B 0,C 180,E1 -3363.184,E2 -3363.184} C_VEL
LIN {X 0,Y 552.111,Z 576.708,A -85,B 0,C 180,E1 -3365.841,E2 -3365.841} C_VEL
LIN {X 0,Y 552.122,Z 576.708,A -85,B 0,C 180,E1 -3369.061,E2 -3369.061} C_VEL
LIN {X 0,Y 552.136,Z 576.704,A -85,B 0,C 180,E1 -3371.443,E2 -3371.443} C_VEL
LIN {X 0,Y 552.091,Z 576.718,A -85,B 0,C 180,E1 -3374.531,E2 -3374.531} C_VEL
LIN {X 0,Y 552.126,Z 576.705,A -85,B 0,C 180,E1 -3377.584,E2 -3377.584} C_VEL
LIN {X 0,Y 552.146,Z 576.711,A -85,B 0,C 180,E1 -3380.474,E2 -3380.474} C_VEL
LIN {X 0,Y 552.109,Z 576.706,A -85,B 0,C 180,E1 -3383.315,E2 -3383.315} C_VEL
LIN {X 0,Y 552.134,Z 576.706,A -85,B 0,C 180,E1 -3385.939,E2 -3385.939} C_VEL
LIN {X 0,Y 552.112,Z 576.714,A -85,B 0,C 180,E1 -3388.54,E2 -3388.54} C_VEL
LIN {X 0,Y 552.119,Z 576.704,A -85,B 0,C 180,E1 -3391.437,E2 -3391.437} C_VEL
LIN {X 0,Y 552.131,Z 576.711,A -85,B 0,C 180,E1 -3394.356,E2 -3394.356} C_VEL
LIN {X 0,Y 552.103,Z 576.711,A -85,B 0,C 180,E1 -3396.758,E2 -3396.758} C_VEL
LIN {X 0,Y 552.113,Z 576.706,A -85,B 0,C 180,E1 -3399.119,E2 -3399.119} C_VEL
LIN {X 0,Y 552.124,Z 576.705,A -85,B 0,C 180,E1 -3401.444,E2 -3401.444} C_VEL
LIN {X 0,Y 552.11,Z 576.708,A -85,B 0,C 180,E1 -3403.737,E2 -3403.737} C_VEL
LIN {X 0,Y 552.129,Z 576.708,A -85,B 0,C 180,E1 -3406.004,E2 -3406.004} C_VEL
LIN {X 0,Y 552.155,Z 576.702,A -85,B 0,C 180,E1 -3408.993,E2 -3408.993} C_VEL
LIN {X 0,Y 552.156,Z 576.705,A -85,B 0,C 180,E1 -3411.951,E2 -3411.951} C_VEL
LIN {X 0,Y 552.226,Z 576.694,A -85,B 0,C 180,E1 -3414.889,E2 -3414.889} C_VEL
LIN {X 0,Y 552.216,Z 576.696,A -85,B 0,C 180,E1 -3417.812,E2 -3417.812} C_VEL
LIN {X 0,Y 552.238,Z 576.694,A -85,B 0,C 180,E1 -3420.729,E2 -3420.729} C_VEL
LIN {X 0,Y 552.203,Z 576.697,A -85,B 0,C 180,E1 -3422.918,E2 -3422.918} C_VEL
LIN {X 0,Y 552.2,Z 576.699,A -85,B 0,C 180,E1 -3425.844,E2 -3425.844} C_VEL
LIN {X 0,Y 552.164,Z 576.703,A -85,B 0,C 180,E1 -3428.785,E2 -3428.785} C_VEL
LIN {X 0,Y 552.157,Z 576.703,A -85,B 0,C 180,E1 -3431.751,E2 -3431.751} C_VEL
LIN {X 0,Y 552.128,Z 576.711,A -85,B 0,C 180,E1 -3434.749,E2 -3434.749} C_VEL
LIN {X 0,Y 552.218,Z 576.841,A -85,B 0,C 180,E1 -3437.266,E2 -3437.266} C_VEL
LIN {X 0,Y 552.222,Z 587.029,A -85,B 0,C 180,E1 -3439.323,E2 -3439.323} C_VEL
LIN {X 0,Y 552.132,Z 593.843,A -85,B 0,C 180,E1 -3440.685,E2 -3440.685} C_VEL
LIN {X 0,Y 553.404,Z 601.478,A -85,B 0,C 180,E1 -3440.829,E2 -3440.829} C_VEL
LIN {X 0,Y 553.171,Z 682.783,A -85,B 0,C 180,E1 -3441.888,E2 -3441.888} C_VEL
LIN {X 0,Y 552.417,Z 688.661,A -85,B 0,C 180,E1 -3441.944,E2 -3441.944} C_VEL
LIN {X 0,Y 549.318,Z 698.162,A -85,B 0,C 180,E1 -3442.006,E2 -3442.006} C_VEL
LIN {X 0,Y 546.486,Z 707.567,A -85,B 0,C 180,E1 -3442.137,E2 -3442.137} C_VEL
LIN {X 0,Y 546.084,Z 713.189,A -85,B 0,C 180,E1 -3442.293,E2 -3442.293} C_VEL
LIN {X 0,Y 545.887,Z 725.091,A -85,B 0,C 180,E1 -3442.72,E2 -3442.72} C_VEL
LIN {X 0,Y 545.687,Z 737.41,A -85,B 0,C 180,E1 -3443.33,E2 -3443.33} C_VEL
LIN {X 0,Y 545.478,Z 749.485,A -85,B 0,C 180,E1 -3444.109,E2 -3444.109} C_VEL
LIN {X 0,Y 545.245,Z 760.029,A -85,B 0,C 180,E1 -3444.969,E2 -3444.969} C_VEL
LIN {X 0,Y 545.053,Z 770.204,A -85,B 0,C 180,E1 -3446.002,E2 -3446.002} C_VEL
LIN {X 0,Y 544.92,Z 779.145,A -85,B 0,C 180,E1 -3447.14,E2 -3447.14} C_VEL
LIN {X 0,Y 544.822,Z 786.442,A -85,B 0,C 180,E1 -3448.298,E2 -3448.298} C_VEL
LIN {X 0,Y 544.718,Z 791.798,A -85,B 0,C 180,E1 -3449.359,E2 -3449.359} C_VEL
LIN {X 0,Y 544.651,Z 796.819,A -85,B 0,C 180,E1 -3450.643,E2 -3450.643} C_VEL
LIN {X 0,Y 544.582,Z 800.476,A -85,B 0,C 180,E1 -3451.946,E2 -3451.946} C_VEL
LIN {X 0,Y 544.569,Z 802.434,A -85,B 0,C 180,E1 -3452.982,E2 -3452.982} C_VEL
LIN {X 0,Y 544.563,Z 803.79,A -85,B 0,C 180,E1 -3454.315,E2 -3454.315} C_VEL
LIN {X 0,Y 544.548,Z 803.886,A -85,B 0,C 180,E1 -3455.603,E2 -3455.603} C_VEL
LIN {X 0,Y 544.562,Z 802.803,A -85,B 0,C 180,E1 -3456.857,E2 -3456.857} C_VEL
LIN {X 0,Y 544.563,Z 800.159,A -85,B 0,C 180,E1 -3458.278,E2 -3458.278} C_VEL
LIN {X 0,Y 544.645,Z 795.959,A -85,B 0,C 180,E1 -3459.697,E2 -3459.697} C_VEL
LIN {X 0,Y 544.703,Z 791.675,A -85,B 0,C 180,E1 -3460.758,E2 -3460.758} C_VEL
LIN {X 0,Y 544.761,Z 786.298,A -85,B 0,C 180,E1 -3461.817,E2 -3461.817} C_VEL
LIN {X 0,Y 544.872,Z 779.877,A -85,B 0,C 180,E1 -3462.845,E2 -3462.845} C_VEL
LIN {X 0,Y 545.025,Z 771.639,A -85,B 0,C 180,E1 -3463.921,E2 -3463.921} C_VEL
LIN {X 0,Y 545.19,Z 762.956,A -85,B 0,C 180,E1 -3464.848,E2 -3464.848} C_VEL
LIN {X 0,Y 545.426,Z 752.523,A -85,B 0,C 180,E1 -3465.751,E2 -3465.751} C_VEL
LIN {X 0,Y 545.623,Z 740.762,A -85,B 0,C 180,E1 -3466.564,E2 -3466.564} C_VEL
LIN {X 0,Y 545.861,Z 728.584,A -85,B 0,C 180,E1 -3467.212,E2 -3467.212} C_VEL
LIN {X 0,Y 546.041,Z 716.995,A -85,B 0,C 180,E1 -3467.679,E2 -3467.679} C_VEL
LIN {X 0,Y 546.154,Z 704.19,A -85,B 0,C 180,E1 -3468.043,E2 -3468.043} C_VEL
LIN {X 0,Y 546.265,Z 687.668,A -85,B 0,C 180,E1 -3468.307,E2 -3468.307} C_VEL
LIN {X 0,Y 546.462,Z 601.521,A -85,B 0,C 180,E1 -3469.444,E2 -3469.444} C_VEL
LIN {X 0,Y 545.117,Z 593.814,A -85,B 0,C 180,E1 -3469.6,E2 -3469.6} C_VEL
LIN {X 0,Y 545.306,Z 579.555,A -85,B 0,C 180,E1 -3472.499,E2 -3472.499} C_VEL
LIN {X 0,Y 545.16,Z 577.578,A -85,B 0,C 180,E1 -3472.919,E2 -3472.919} C_VEL
LIN {X 0,Y 545.075,Z 577.587,A -85,B 0,C 180,E1 -3476.33,E2 -3476.33} C_VEL
LIN {X 0,Y 545.063,Z 577.584,A -85,B 0,C 180,E1 -3478.953,E2 -3478.953} C_VEL
LIN {X 0,Y 545.102,Z 577.581,A -85,B 0,C 180,E1 -3481.509,E2 -3481.509} C_VEL
LIN {X 0,Y 545.093,Z 577.583,A -85,B 0,C 180,E1 -3484.492,E2 -3484.492} C_VEL
LIN {X 0,Y 545.043,Z 577.586,A -85,B 0,C 180,E1 -3487.244,E2 -3487.244} C_VEL
LIN {X 0,Y 545.12,Z 577.583,A -85,B 0,C 180,E1 -3490.416,E2 -3490.416} C_VEL
LIN {X 0,Y 545.074,Z 577.583,A -85,B 0,C 180,E1 -3493.522,E2 -3493.522} C_VEL
LIN {X 0,Y 545.096,Z 577.582,A -85,B 0,C 180,E1 -3495.821,E2 -3495.821} C_VEL
LIN {X 0,Y 545.118,Z 577.579,A -85,B 0,C 180,E1 -3498.85,E2 -3498.85} C_VEL
LIN {X 0,Y 545.13,Z 577.577,A -85,B 0,C 180,E1 -3501.848,E2 -3501.848} C_VEL
LIN {X 0,Y 545.203,Z 577.57,A -85,B 0,C 180,E1 -3504.824,E2 -3504.824} C_VEL
LIN {X 0,Y 545.198,Z 577.567,A -85,B 0,C 180,E1 -3507.785,E2 -3507.785} C_VEL
LIN {X 0,Y 545.215,Z 577.572,A -85,B 0,C 180,E1 -3510.739,E2 -3510.739} C_VEL
LIN {X 0,Y 545.176,Z 577.574,A -85,B 0,C 180,E1 -3512.957,E2 -3512.957} C_VEL
LIN {X 0,Y 545.172,Z 577.57,A -85,B 0,C 180,E1 -3515.92,E2 -3515.92} C_VEL
LIN {X 0,Y 545.124,Z 577.583,A -85,B 0,C 180,E1 -3518.901,E2 -3518.901} C_VEL
LIN {X 0,Y 545.139,Z 577.574,A -85,B 0,C 180,E1 -3521.905,E2 -3521.905} C_VEL
LIN {X 0,Y 545.089,Z 577.588,A -85,B 0,C 180,E1 -3524.944,E2 -3524.944} C_VEL
LIN {X 0,Y 545.081,Z 577.581,A -85,B 0,C 180,E1 -3528.026,E2 -3528.026} C_VEL
LIN {X 0,Y 545.097,Z 577.581,A -85,B 0,C 180,E1 -3530.373,E2 -3530.373} C_VEL
LIN {X 0,Y 545.082,Z 577.583,A -85,B 0,C 180,E1 -3533.56,E2 -3533.56} C_VEL
LIN {X 0,Y 545.084,Z 577.581,A -85,B 0,C 180,E1 -3536.001,E2 -3536.001} C_VEL
LIN {X 0,Y 545.093,Z 577.584,A -85,B 0,C 180,E1 -3538.749,E2 -3538.749} C_VEL
LIN {X 0,Y 545.062,Z 577.586,A -85,B 0,C 180,E1 -3541.679,E2 -3541.679} C_VEL
LIN {X 0,Y 545.08,Z 577.583,A -85,B 0,C 180,E1 -3544.564,E2 -3544.564} C_VEL
LIN {X 0,Y 545.041,Z 577.595,A -85,B 0,C 180,E1 -3547.304,E2 -3547.304} C_VEL
LIN {X 0,Y 545.072,Z 577.582,A -85,B 0,C 180,E1 -3550.143,E2 -3550.143} C_VEL
LIN {X 0,Y 545.082,Z 577.587,A -85,B 0,C 180,E1 -3553.107,E2 -3553.107} C_VEL
LIN {X 0,Y 545.071,Z 577.583,A -85,B 0,C 180,E1 -3556.225,E2 -3556.225} C_VEL
LIN {X 0,Y 545.091,Z 577.582,A -85,B 0,C 180,E1 -3558.886,E2 -3558.886} C_VEL
LIN {X 0,Y 545.057,Z 577.59,A -85,B 0,C 180,E1 -3561.763,E2 -3561.763} C_VEL
LIN {X 0,Y 545.041,Z 577.586,A -85,B 0,C 180,E1 -3564.532,E2 -3564.532} C_VEL
LIN {X 0,Y 545.074,Z 577.586,A -85,B 0,C 180,E1 -3567.212,E2 -3567.212} C_VEL
LIN {X 0,Y 545.068,Z 577.59,A -85,B 0,C 180,E1 -3569.811,E2 -3569.811} C_VEL
LIN {X 0,Y 545.086,Z 577.582,A -85,B 0,C 180,E1 -3572.344,E2 -3572.344} C_VEL
LIN {X 0,Y 545.122,Z 577.576,A -85,B 0,C 180,E1 -3574.821,E2 -3574.821} C_VEL
LIN {X 0,Y 545.041,Z 577.588,A -85,B 0,C 180,E1 -3577.242,E2 -3577.242} C_VEL
LIN {X 0,Y 545.121,Z 577.578,A -85,B 0,C 180,E1 -3580.415,E2 -3580.415} C_VEL
LIN {X 0,Y 545.077,Z 577.586,A -85,B 0,C 180,E1 -3583.521,E2 -3583.521} C_VEL
LIN {X 0,Y 545.1,Z 577.587,A -85,B 0,C 180,E1 -3585.82,E2 -3585.82} C_VEL
LIN {X 0,Y 545.123,Z 577.576,A -85,B 0,C 180,E1 -3588.85,E2 -3588.85} C_VEL
LIN {X 0,Y 545.131,Z 577.582,A -85,B 0,C 180,E1 -3591.847,E2 -3591.847} C_VEL
LIN {X 0,Y 545.209,Z 577.566,A -85,B 0,C 180,E1 -3594.823,E2 -3594.823} C_VEL
LIN {X 0,Y 545.201,Z 577.57,A -85,B 0,C 180,E1 -3597.784,E2 -3597.784} C_VEL
LIN {X 0,Y 545.217,Z 577.566,A -85,B 0,C 180,E1 -3600.739,E2 -3600.739} C_VEL
LIN {X 0,Y 545.177,Z 577.57,A -85,B 0,C 180,E1 -3602.956,E2 -3602.956} C_VEL
LIN {X 0,Y 545.172,Z 577.574,A -85,B 0,C 180,E1 -3605.92,E2 -3605.92} C_VEL
LIN {X 0,Y 545.116,Z 577.579,A -85,B 0,C 180,E1 -3608.9,E2 -3608.9} C_VEL
LIN {X 0,Y 545.14,Z 577.576,A -85,B 0,C 180,E1 -3611.904,E2 -3611.904} C_VEL
LIN {X 0,Y 545.091,Z 577.583,A -85,B 0,C 180,E1 -3614.944,E2 -3614.944} C_VEL
LIN {X 0,Y 545.078,Z 577.584,A -85,B 0,C 180,E1 -3618.026,E2 -3618.026} C_VEL
LIN {X 0,Y 545.098,Z 577.586,A -85,B 0,C 180,E1 -3620.372,E2 -3620.372} C_VEL
LIN {X 0,Y 545.084,Z 577.581,A -85,B 0,C 180,E1 -3623.559,E2 -3623.559} C_VEL
LIN {X 0,Y 545.084,Z 577.582,A -85,B 0,C 180,E1 -3626.001,E2 -3626.001} C_VEL
LIN {X 0,Y 545.095,Z 577.589,A -85,B 0,C 180,E1 -3628.748,E2 -3628.748} C_VEL
LIN {X 0,Y 545.063,Z 577.583,A -85,B 0,C 180,E1 -3631.679,E2 -3631.679} C_VEL
LIN {X 0,Y 545.078,Z 577.587,A -85,B 0,C 180,E1 -3634.564,E2 -3634.564} C_VEL
LIN {X 0,Y 545.042,Z 577.589,A -85,B 0,C 180,E1 -3637.304,E2 -3637.304} C_VEL
LIN {X 0,Y 545.072,Z 577.583,A -85,B 0,C 180,E1 -3640.142,E2 -3640.142} C_VEL
LIN {X 0,Y 545.084,Z 577.589,A -85,B 0,C 180,E1 -3643.106,E2 -3643.106} C_VEL
LIN {X 0,Y 545.054,Z 577.585,A -85,B 0,C 180,E1 -3646.226,E2 -3646.226} C_VEL
LIN {X 0,Y 545.087,Z 577.587,A -85,B 0,C 180,E1 -3648.885,E2 -3648.885} C_VEL
LIN {X 0,Y 545.088,Z 577.586,A -85,B 0,C 180,E1 -3650.818,E2 -3650.818} C_VEL
LIN {X 0,Y 545.048,Z 577.588,A -85,B 0,C 180,E1 -3653.619,E2 -3653.619} C_VEL
LIN {X 0,Y 545.076,Z 577.583,A -85,B 0,C 180,E1 -3656.328,E2 -3656.328} C_VEL
LIN {X 0,Y 545.07,Z 577.588,A -85,B 0,C 180,E1 -3658.952,E2 -3658.952} C_VEL
LIN {X 0,Y 545.107,Z 577.587,A -85,B 0,C 180,E1 -3661.507,E2 -3661.507} C_VEL
LIN {X 0,Y 545.1,Z 577.584,A -85,B 0,C 180,E1 -3664.491,E2 -3664.491} C_VEL
LIN {X 0,Y 545.143,Z 577.688,A -85,B 0,C 180,E1 -3664.923,E2 -3664.923} C_VEL
LIN {X 0,Y 546.46,Z 584.314,A -85,B 0,C 180,E1 -3665.942,E2 -3665.942} C_VEL
LIN {X 0,Y 546.474,Z 595.013,A -85,B 0,C 180,E1 -3667.483,E2 -3667.483} C_VEL
LIN {X 0,Y 546.066,Z 614.674,A -85,B 0,C 180,E1 -3670.266,E2 -3670.266} C_VEL
LIN {X 0,Y 545.699,Z 635.058,A -85,B 0,C 180,E1 -3673.155,E2 -3673.155} C_VEL
LIN {X 0,Y 545.431,Z 651.336,A -85,B 0,C 180,E1 -3675.433,E2 -3675.433} C_VEL
LIN {X 0,Y 546.539,Z 659.869,A -85,B 0,C 180,E1 -3675.581,E2 -3675.581} C_VEL
LIN {X 0,Y 546.253,Z 759.91,A -85,B 0,C 180,E1 -3676.917,E2 -3676.917} C_VEL
LIN {X 0,Y 546.06,Z 773.194,A -85,B 0,C 180,E1 -3677.243,E2 -3677.243} C_VEL
LIN {X 0,Y 545.903,Z 786.47,A -85,B 0,C 180,E1 -3677.735,E2 -3677.735} C_VEL
LIN {X 0,Y 545.729,Z 798.354,A -85,B 0,C 180,E1 -3678.341,E2 -3678.341} C_VEL
LIN {X 0,Y 545.498,Z 809.187,A -85,B 0,C 180,E1 -3679.045,E2 -3679.045} C_VEL
LIN {X 0,Y 545.259,Z 819.595,A -85,B 0,C 180,E1 -3679.885,E2 -3679.885} C_VEL
LIN {X 0,Y 545.085,Z 828.106,A -85,B 0,C 180,E1 -3680.725,E2 -3680.725} C_VEL
LIN {X 0,Y 544.976,Z 835.955,A -85,B 0,C 180,E1 -3681.657,E2 -3681.657} C_VEL
LIN {X 0,Y 544.825,Z 843.617,A -85,B 0,C 180,E1 -3682.774,E2 -3682.774} C_VEL
LIN {X 0,Y 544.777,Z 850.676,A -85,B 0,C 180,E1 -3684.075,E2 -3684.075} C_VEL
LIN {X 0,Y 544.629,Z 855.37,A -85,B 0,C 180,E1 -3685.188,E2 -3685.188} C_VEL
LIN {X 0,Y 544.669,Z 858.956,A -85,B 0,C 180,E1 -3686.3,E2 -3686.3} C_VEL
LIN {X 0,Y 544.651,Z 860.806,A -85,B 0,C 180,E1 -3687.041,E2 -3687.041} C_VEL
LIN {X 0,Y 544.546,Z 863.183,A -85,B 0,C 180,E1 -3688.52,E2 -3688.52} C_VEL
LIN {X 0,Y 544.541,Z 864,A -85,B 0,C 180,E1 -3689.999,E2 -3689.999} C_VEL
LIN {X 0,Y 544.546,Z 863.186,A -85,B 0,C 180,E1 -3691.478,E2 -3691.478} C_VEL
LIN {X 0,Y 544.65,Z 860.812,A -85,B 0,C 180,E1 -3692.958,E2 -3692.958} C_VEL
LIN {X 0,Y 544.684,Z 857.898,A -85,B 0,C 180,E1 -3694.069,E2 -3694.069} C_VEL
LIN {X 0,Y 544.653,Z 853.952,A -85,B 0,C 180,E1 -3695.181,E2 -3695.181} C_VEL
LIN {X 0,Y 544.729,Z 848.646,A -85,B 0,C 180,E1 -3696.339,E2 -3696.339} C_VEL
LIN {X 0,Y 544.836,Z 842.473,A -85,B 0,C 180,E1 -3697.411,E2 -3697.411} C_VEL
LIN {X 0,Y 545.006,Z 834.484,A -85,B 0,C 180,E1 -3698.527,E2 -3698.527} C_VEL
LIN {X 0,Y 545.151,Z 826.343,A -85,B 0,C 180,E1 -3699.46,E2 -3699.46} C_VEL
LIN {X 0,Y 545.372,Z 816.409,A -85,B 0,C 180,E1 -3700.393,E2 -3700.393} C_VEL
LIN {X 0,Y 545.552,Z 805.552,A -85,B 0,C 180,E1 -3701.211,E2 -3701.211} C_VEL
LIN {X 0,Y 545.765,Z 794.19,A -85,B 0,C 180,E1 -3701.889,E2 -3701.889} C_VEL
LIN {X 0,Y 545.925,Z 781.997,A -85,B 0,C 180,E1 -3702.452,E2 -3702.452} C_VEL
LIN {X 0,Y 546.079,Z 769.209,A -85,B 0,C 180,E1 -3702.873,E2 -3702.873} C_VEL
LIN {X 0,Y 546.258,Z 755.658,A -85,B 0,C 180,E1 -3703.153,E2 -3703.153} C_VEL
LIN {X 0,Y 546.508,Z 658.206,A -85,B 0,C 180,E1 -3704.442,E2 -3704.442} C_VEL
LIN {X 0,Y 545.443,Z 651.325,A -85,B 0,C 180,E1 -3704.568,E2 -3704.568} C_VEL
LIN {X 0,Y 545.8,Z 630.206,A -85,B 0,C 180,E1 -3707.528,E2 -3707.528} C_VEL
LIN {X 0,Y 546.186,Z 609.044,A -85,B 0,C 180,E1 -3710.525,E2 -3710.525} C_VEL
LIN {X 0,Y 546.551,Z 587.975,A -85,B 0,C 180,E1 -3713.491,E2 -3713.491} C_VEL
LIN {X 0,Y 546.436,Z 584.072,A -85,B 0,C 180,E1 -3714.053,E2 -3714.053} C_VEL
LIN {X 0,Y 545.105,Z 577.586,A -85,B 0,C 180,E1 -3715.077,E2 -3715.077} C_VEL
LIN {X 0,Y 545.091,Z 577.583,A -85,B 0,C 180,E1 -3717.655,E2 -3717.655} C_VEL
LIN {X 0,Y 545.075,Z 577.589,A -85,B 0,C 180,E1 -3720.245,E2 -3720.245} C_VEL
LIN {X 0,Y 545.087,Z 577.585,A -85,B 0,C 180,E1 -3723.063,E2 -3723.063} C_VEL
LIN {X 0,Y 545.061,Z 577.586,A -85,B 0,C 180,E1 -3725.676,E2 -3725.676} C_VEL
LIN {X 0,Y 545.051,Z 577.592,A -85,B 0,C 180,E1 -3728.236,E2 -3728.236} C_VEL
LIN {X 0,Y 545.097,Z 577.583,A -85,B 0,C 180,E1 -3731.112,E2 -3731.112} C_VEL
LIN {X 0,Y 545.054,Z 577.591,A -85,B 0,C 180,E1 -3734.128,E2 -3734.128} C_VEL
LIN {X 0,Y 545.082,Z 577.586,A -85,B 0,C 180,E1 -3736.893,E2 -3736.893} C_VEL
LIN {X 0,Y 545.09,Z 577.583,A -85,B 0,C 180,E1 -3739.859,E2 -3739.859} C_VEL
LIN {X 0,Y 545.07,Z 577.584,A -85,B 0,C 180,E1 -3743.072,E2 -3743.072} C_VEL
LIN {X 0,Y 545.084,Z 577.582,A -85,B 0,C 180,E1 -3745.605,E2 -3745.605} C_VEL
LIN {X 0,Y 545.072,Z 577.591,A -85,B 0,C 180,E1 -3748.317,E2 -3748.317} C_VEL
LIN {X 0,Y 545.086,Z 577.58,A -85,B 0,C 180,E1 -3751.25,E2 -3751.25} C_VEL
LIN {X 0,Y 545.083,Z 577.584,A -85,B 0,C 180,E1 -3753.999,E2 -3753.999} C_VEL
LIN {X 0,Y 545.085,Z 577.589,A -85,B 0,C 180,E1 -3756.441,E2 -3756.441} C_VEL
LIN {X 0,Y 545.088,Z 577.581,A -85,B 0,C 180,E1 -3759.627,E2 -3759.627} C_VEL
LIN {X 0,Y 545.087,Z 577.586,A -85,B 0,C 180,E1 -3762.75,E2 -3762.75} C_VEL
LIN {X 0,Y 545.088,Z 577.583,A -85,B 0,C 180,E1 -3765.82,E2 -3765.82} C_VEL
LIN {X 0,Y 545.11,Z 577.581,A -85,B 0,C 180,E1 -3768.849,E2 -3768.849} C_VEL
LIN {X 0,Y 545.126,Z 577.579,A -85,B 0,C 180,E1 -3771.847,E2 -3771.847} C_VEL
LIN {X 0,Y 545.201,Z 577.57,A -85,B 0,C 180,E1 -3774.823,E2 -3774.823} C_VEL
LIN {X 0,Y 545.188,Z 577.571,A -85,B 0,C 180,E1 -3777.784,E2 -3777.784} C_VEL
LIN {X 0,Y 545.208,Z 577.57,A -85,B 0,C 180,E1 -3780.738,E2 -3780.738} C_VEL
LIN {X 0,Y 545.169,Z 577.573,A -85,B 0,C 180,E1 -3782.956,E2 -3782.956} C_VEL
LIN {X 0,Y 545.172,Z 577.576,A -85,B 0,C 180,E1 -3785.919,E2 -3785.919} C_VEL
LIN {X 0,Y 545.121,Z 577.58,A -85,B 0,C 180,E1 -3788.9,E2 -3788.9} C_VEL
LIN {X 0,Y 545.128,Z 577.581,A -85,B 0,C 180,E1 -3791.904,E2 -3791.904} C_VEL
LIN {X 0,Y 545.078,Z 577.588,A -85,B 0,C 180,E1 -3794.944,E2 -3794.944} C_VEL
LIN {X 0,Y 545.158,Z 577.674,A -85,B 0,C 180,E1 -3797.2,E2 -3797.2} C_VEL
LIN {X 0,Y 545.212,Z 585.478,A -85,B 0,C 180,E1 -3798.8,E2 -3798.8} C_VEL
LIN {X 0,Y 545.065,Z 593.853,A -85,B 0,C 180,E1 -3800.496,E2 -3800.496} C_VEL
LIN {X 0,Y 546.539,Z 602.444,A -85,B 0,C 180,E1 -3800.66,E2 -3800.66} C_VEL
LIN {X 0,Y 546.195,Z 700.226,A -85,B 0,C 180,E1 -3801.967,E2 -3801.967} C_VEL
LIN {X 0,Y 546.084,Z 713.189,A -85,B 0,C 180,E1 -3802.293,E2 -3802.293} C_VEL
LIN {X 0,Y 545.865,Z 716.976,A -85,B 0,C 180,E1 -3802.411,E2 -3802.411} C_VEL
LIN {X 0,Y 543.956,Z 724.411,A -85,B 0,C 180,E1 -3802.648,E2 -3802.648} C_VEL
LIN {X 0,Y 539.44,Z 736.638,A -85,B 0,C 180,E1 -3803.147,E2 -3803.147} C_VEL
LIN {X 0,Y 538.636,Z 741.748,A -85,B 0,C 180,E1 -3803.437,E2 -3803.437} C_VEL
LIN {X 0,Y 538.403,Z 752.485,A -85,B 0,C 180,E1 -3804.195,E2 -3804.195} C_VEL
LIN {X 0,Y 538.2,Z 762.946,A -85,B 0,C 180,E1 -3805.112,E2 -3805.112} C_VEL
LIN {X 0,Y 537.957,Z 772.695,A -85,B 0,C 180,E1 -3806.18,E2 -3806.18} C_VEL
LIN {X 0,Y 537.828,Z 780.996,A -85,B 0,C 180,E1 -3807.307,E2 -3807.307} C_VEL
LIN {X 0,Y 537.696,Z 787.811,A -85,B 0,C 180,E1 -3808.464,E2 -3808.464} C_VEL
LIN {X 0,Y 537.582,Z 793.918,A -85,B 0,C 180,E1 -3809.788,E2 -3809.788} C_VEL
LIN {X 0,Y 537.547,Z 798.395,A -85,B 0,C 180,E1 -3811.093,E2 -3811.093} C_VEL
LIN {X 0,Y 537.466,Z 801.538,A -85,B 0,C 180,E1 -3812.42,E2 -3812.42} C_VEL
LIN {X 0,Y 537.457,Z 802.941,A -85,B 0,C 180,E1 -3813.313,E2 -3813.313} C_VEL
LIN {X 0,Y 537.462,Z 803.9,A -85,B 0,C 180,E1 -3814.534,E2 -3814.534} C_VEL
LIN {X 0,Y 537.44,Z 803.761,A -85,B 0,C 180,E1 -3815.831,E2 -3815.831} C_VEL
LIN {X 0,Y 537.455,Z 802.492,A -85,B 0,C 180,E1 -3817.094,E2 -3817.094} C_VEL
LIN {X 0,Y 537.468,Z 800.151,A -85,B 0,C 180,E1 -3818.321,E2 -3818.321} C_VEL
LIN {X 0,Y 537.533,Z 796.763,A -85,B 0,C 180,E1 -3819.522,E2 -3819.522} C_VEL
LIN {X 0,Y 537.62,Z 791.758,A -85,B 0,C 180,E1 -3820.815,E2 -3820.815} C_VEL
LIN {X 0,Y 537.694,Z 785.444,A -85,B 0,C 180,E1 -3822.056,E2 -3822.056} C_VEL
LIN {X 0,Y 537.84,Z 778.58,A -85,B 0,C 180,E1 -3823.136,E2 -3823.136} C_VEL
LIN {X 0,Y 538.016,Z 770.087,A -85,B 0,C 180,E1 -3824.221,E2 -3824.221} C_VEL
LIN {X 0,Y 538.259,Z 759.782,A -85,B 0,C 180,E1 -3825.276,E2 -3825.276} C_VEL
LIN {X 0,Y 538.484,Z 748.867,A -85,B 0,C 180,E1 -3826.17,E2 -3826.17} C_VEL
LIN {X 0,Y 538.759,Z 737.122,A -85,B 0,C 180,E1 -3826.929,E2 -3826.929} C_VEL
LIN {X 0,Y 538.957,Z 725.964,A -85,B 0,C 180,E1 -3827.493,E2 -3827.493} C_VEL
LIN {X 0,Y 539.17,Z 713.075,A -85,B 0,C 180,E1 -3827.972,E2 -3827.972} C_VEL
LIN {X 0,Y 539.302,Z 700.251,A -85,B 0,C 180,E1 -3828.293,E2 -3828.293} C_VEL
LIN {X 0,Y 539.482,Z 601.667,A -85,B 0,C 180,E1 -3829.633,E2 -3829.633} C_VEL
LIN {X 0,Y 538.096,Z 593.867,A -85,B 0,C 180,E1 -3829.783,E2 -3829.783} C_VEL
LIN {X 0,Y 538.312,Z 580.799,A -85,B 0,C 180,E1 -3832.521,E2 -3832.521} C_VEL
LIN {X 0,Y 538.09,Z 578.46,A -85,B 0,C 180,E1 -3833.074,E2 -3833.074} C_VEL
LIN {X 0,Y 538.03,Z 578.469,A -85,B 0,C 180,E1 -3835.829,E2 -3835.829} C_VEL
LIN {X 0,Y 538.006,Z 578.465,A -85,B 0,C 180,E1 -3838.5,E2 -3838.5} C_VEL
LIN {X 0,Y 538.057,Z 578.456,A -85,B 0,C 180,E1 -3841.101,E2 -3841.101} C_VEL
LIN {X 0,Y 538.04,Z 578.462,A -85,B 0,C 180,E1 -3843.634,E2 -3843.634} C_VEL
LIN {X 0,Y 538.021,Z 578.471,A -85,B 0,C 180,E1 -3846.119,E2 -3846.119} C_VEL
LIN {X 0,Y 538.038,Z 578.459,A -85,B 0,C 180,E1 -3849.35,E2 -3849.35} C_VEL
LIN {X 0,Y 538.073,Z 578.459,A -85,B 0,C 180,E1 -3852.519,E2 -3852.519} C_VEL
LIN {X 0,Y 538.065,Z 578.456,A -85,B 0,C 180,E1 -3855.632,E2 -3855.632} C_VEL
LIN {X 0,Y 538.077,Z 578.458,A -85,B 0,C 180,E1 -3858.702,E2 -3858.702} C_VEL
LIN {X 0,Y 538.087,Z 578.454,A -85,B 0,C 180,E1 -3861.74,E2 -3861.74} C_VEL
LIN {X 0,Y 538.161,Z 578.448,A -85,B 0,C 180,E1 -3864.756,E2 -3864.756} C_VEL
LIN {X 0,Y 538.17,Z 578.443,A -85,B 0,C 180,E1 -3867.756,E2 -3867.756} C_VEL
LIN {X 0,Y 538.185,Z 578.447,A -85,B 0,C 180,E1 -3870.749,E2 -3870.749} C_VEL
LIN {X 0,Y 538.143,Z 578.449,A -85,B 0,C 180,E1 -3872.995,E2 -3872.995} C_VEL
LIN {X 0,Y 538.126,Z 578.449,A -85,B 0,C 180,E1 -3875.998,E2 -3875.998} C_VEL
LIN {X 0,Y 538.075,Z 578.459,A -85,B 0,C 180,E1 -3879.018,E2 -3879.018} C_VEL
LIN {X 0,Y 538.087,Z 578.453,A -85,B 0,C 180,E1 -3882.063,E2 -3882.063} C_VEL
LIN {X 0,Y 538.049,Z 578.462,A -85,B 0,C 180,E1 -3885.144,E2 -3885.144} C_VEL
LIN {X 0,Y 538.033,Z 578.461,A -85,B 0,C 180,E1 -3888.271,E2 -3888.271} C_VEL
LIN {X 0,Y 538.042,Z 578.464,A -85,B 0,C 180,E1 -3890.652,E2 -3890.652} C_VEL
LIN {X 0,Y 538.006,Z 578.463,A -85,B 0,C 180,E1 -3893.889,E2 -3893.889} C_VEL
LIN {X 0,Y 538.046,Z 578.459,A -85,B 0,C 180,E1 -3896.367,E2 -3896.367} C_VEL
LIN {X 0,Y 538.035,Z 578.467,A -85,B 0,C 180,E1 -3898.934,E2 -3898.934} C_VEL
LIN {X 0,Y 538.014,Z 578.462,A -85,B 0,C 180,E1 -3901.888,E2 -3901.888} C_VEL
LIN {X 0,Y 538.029,Z 578.462,A -85,B 0,C 180,E1 -3904.62,E2 -3904.62} C_VEL
LIN {X 0,Y 538.009,Z 578.472,A -85,B 0,C 180,E1 -3907.17,E2 -3907.17} C_VEL
LIN {X 0,Y 538.03,Z 578.462,A -85,B 0,C 180,E1 -3909.797,E2 -3909.797} C_VEL
LIN {X 0,Y 538.023,Z 578.463,A -85,B 0,C 180,E1 -3912.786,E2 -3912.786} C_VEL
LIN {X 0,Y 538.033,Z 578.461,A -85,B 0,C 180,E1 -3915.926,E2 -3915.926} C_VEL
LIN {X 0,Y 538.053,Z 578.464,A -85,B 0,C 180,E1 -3919.253,E2 -3919.253} C_VEL
LIN {X 0,Y 537.997,Z 578.465,A -85,B 0,C 180,E1 -3922.123,E2 -3922.123} C_VEL
LIN {X 0,Y 538.003,Z 578.464,A -85,B 0,C 180,E1 -3924.916,E2 -3924.916} C_VEL
LIN {X 0,Y 538.023,Z 578.471,A -85,B 0,C 180,E1 -3927.618,E2 -3927.618} C_VEL
LIN {X 0,Y 538.022,Z 578.462,A -85,B 0,C 180,E1 -3930.239,E2 -3930.239} C_VEL
LIN {X 0,Y 538.062,Z 578.456,A -85,B 0,C 180,E1 -3932.796,E2 -3932.796} C_VEL
LIN {X 0,Y 538.032,Z 578.462,A -85,B 0,C 180,E1 -3935.292,E2 -3935.292} C_VEL
LIN {X 0,Y 538.02,Z 578.467,A -85,B 0,C 180,E1 -3938.042,E2 -3938.042} C_VEL
LIN {X 0,Y 538.037,Z 578.459,A -85,B 0,C 180,E1 -3940.94,E2 -3940.94} C_VEL
LIN {X 0,Y 538.024,Z 578.462,A -85,B 0,C 180,E1 -3943.299,E2 -3943.299} C_VEL
LIN {X 0,Y 538.069,Z 578.46,A -85,B 0,C 180,E1 -3945.631,E2 -3945.631} C_VEL
LIN {X 0,Y 538.082,Z 578.454,A -85,B 0,C 180,E1 -3948.702,E2 -3948.702} C_VEL
LIN {X 0,Y 538.088,Z 578.457,A -85,B 0,C 180,E1 -3951.74,E2 -3951.74} C_VEL
LIN {X 0,Y 538.166,Z 578.444,A -85,B 0,C 180,E1 -3954.755,E2 -3954.755} C_VEL
LIN {X 0,Y 538.173,Z 578.446,A -85,B 0,C 180,E1 -3957.755,E2 -3957.755} C_VEL
LIN {X 0,Y 538.187,Z 578.442,A -85,B 0,C 180,E1 -3960.748,E2 -3960.748} C_VEL
LIN {X 0,Y 538.143,Z 578.446,A -85,B 0,C 180,E1 -3962.995,E2 -3962.995} C_VEL
LIN {X 0,Y 538.126,Z 578.453,A -85,B 0,C 180,E1 -3965.997,E2 -3965.997} C_VEL
LIN {X 0,Y 538.066,Z 578.456,A -85,B 0,C 180,E1 -3969.018,E2 -3969.018} C_VEL
LIN {X 0,Y 538.089,Z 578.457,A -85,B 0,C 180,E1 -3972.063,E2 -3972.063} C_VEL
LIN {X 0,Y 538.051,Z 578.458,A -85,B 0,C 180,E1 -3975.144,E2 -3975.144} C_VEL
LIN {X 0,Y 538.032,Z 578.465,A -85,B 0,C 180,E1 -3978.27,E2 -3978.27} C_VEL
LIN {X 0,Y 538.043,Z 578.467,A -85,B 0,C 180,E1 -3980.651,E2 -3980.651} C_VEL
LIN {X 0,Y 538.008,Z 578.463,A -85,B 0,C 180,E1 -3983.888,E2 -3983.888} C_VEL
LIN {X 0,Y 538.046,Z 578.463,A -85,B 0,C 180,E1 -3986.367,E2 -3986.367} C_VEL
LIN {X 0,Y 538.036,Z 578.465,A -85,B 0,C 180,E1 -3988.933,E2 -3988.933} C_VEL
LIN {X 0,Y 538.016,Z 578.461,A -85,B 0,C 180,E1 -3991.887,E2 -3991.887} C_VEL
LIN {X 0,Y 538.027,Z 578.467,A -85,B 0,C 180,E1 -3994.619,E2 -3994.619} C_VEL
LIN {X 0,Y 538.01,Z 578.467,A -85,B 0,C 180,E1 -3997.17,E2 -3997.17} C_VEL
LIN {X 0,Y 538.028,Z 578.46,A -85,B 0,C 180,E1 -3999.797,E2 -3999.797} C_VEL
LIN {X 0,Y 538.025,Z 578.467,A -85,B 0,C 180,E1 -4002.786,E2 -4002.786} C_VEL
LIN {X 0,Y 538.034,Z 578.467,A -85,B 0,C 180,E1 -4005.14,E2 -4005.14} C_VEL
LIN {X 0,Y 538.036,Z 578.459,A -85,B 0,C 180,E1 -4008.226,E2 -4008.226} C_VEL
LIN {X 0,Y 538.02,Z 578.47,A -85,B 0,C 180,E1 -4011.169,E2 -4011.169} C_VEL
LIN {X 0,Y 538.001,Z 578.463,A -85,B 0,C 180,E1 -4014.088,E2 -4014.088} C_VEL
LIN {X 0,Y 538.036,Z 578.462,A -85,B 0,C 180,E1 -4016.727,E2 -4016.727} C_VEL
LIN {X 0,Y 538.02,Z 578.468,A -85,B 0,C 180,E1 -4019.558,E2 -4019.558} C_VEL
LIN {X 0,Y 538.045,Z 578.462,A -85,B 0,C 180,E1 -4021.95,E2 -4021.95} C_VEL
LIN {X 0,Y 538.109,Z 578.609,A -85,B 0,C 180,E1 -4024.753,E2 -4024.753} C_VEL
LIN {X 0,Y 539.591,Z 586.041,A -85,B 0,C 180,E1 -4025.91,E2 -4025.91} C_VEL
LIN {X 0,Y 539.471,Z 598.094,A -85,B 0,C 180,E1 -4027.662,E2 -4027.662} C_VEL
LIN {X 0,Y 539.083,Z 615.72,A -85,B 0,C 180,E1 -4030.186,E2 -4030.186} C_VEL
LIN {X 0,Y 538.756,Z 635.058,A -85,B 0,C 180,E1 -4032.931,E2 -4032.931} C_VEL
LIN {X 0,Y 538.433,Z 651.415,A -85,B 0,C 180,E1 -4035.245,E2 -4035.245} C_VEL
LIN {X 0,Y 539.673,Z 659.784,A -85,B 0,C 180,E1 -4035.392,E2 -4035.392} C_VEL
LIN {X 0,Y 539.332,Z 759.91,A -85,B 0,C 180,E1 -4036.746,E2 -4036.746} C_VEL
LIN {X 0,Y 539.152,Z 773.193,A -85,B 0,C 180,E1 -4037.077,E2 -4037.077} C_VEL
LIN {X 0,Y 538.955,Z 786.471,A -85,B 0,C 180,E1 -4037.574,E2 -4037.574} C_VEL
LIN {X 0,Y 538.747,Z 798.352,A -85,B 0,C 180,E1 -4038.188,E2 -4038.188} C_VEL
LIN {X 0,Y 538.486,Z 810.476,A -85,B 0,C 180,E1 -4038.995,E2 -4038.995} C_VEL
LIN {X 0,Y 538.227,Z 820.638,A -85,B 0,C 180,E1 -4039.846,E2 -4039.846} C_VEL
LIN {X 0,Y 538.027,Z 829.779,A -85,B 0,C 180,E1 -4040.791,E2 -4040.791} C_VEL
LIN {X 0,Y 537.851,Z 838.683,A -85,B 0,C 180,E1 -4041.924,E2 -4041.924} C_VEL
LIN {X 0,Y 537.73,Z 845.844,A -85,B 0,C 180,E1 -4043.055,E2 -4043.055} C_VEL
LIN {X 0,Y 537.677,Z 852.363,A -85,B 0,C 180,E1 -4044.373,E2 -4044.373} C_VEL
LIN {X 0,Y 537.558,Z 856.674,A -85,B 0,C 180,E1 -4045.5,E2 -4045.5} C_VEL
LIN {X 0,Y 537.591,Z 858.956,A -85,B 0,C 180,E1 -4046.251,E2 -4046.251} C_VEL
LIN {X 0,Y 537.551,Z 860.806,A -85,B 0,C 180,E1 -4047.001,E2 -4047.001} C_VEL
LIN {X 0,Y 537.451,Z 863.182,A -85,B 0,C 180,E1 -4048.501,E2 -4048.501} C_VEL
LIN {X 0,Y 537.442,Z 864,A -85,B 0,C 180,E1 -4049.999,E2 -4049.999} C_VEL
LIN {X 0,Y 537.451,Z 863.185,A -85,B 0,C 180,E1 -4051.498,E2 -4051.498} C_VEL
LIN {X 0,Y 537.551,Z 860.812,A -85,B 0,C 180,E1 -4052.997,E2 -4052.997} C_VEL
LIN {X 0,Y 537.603,Z 857.898,A -85,B 0,C 180,E1 -4054.122,E2 -4054.122} C_VEL
LIN {X 0,Y 537.587,Z 853.951,A -85,B 0,C 180,E1 -4055.25,E2 -4055.25} C_VEL
LIN {X 0,Y 537.644,Z 849.127,A -85,B 0,C 180,E1 -4056.326,E2 -4056.326} C_VEL
LIN {X 0,Y 537.79,Z 842.473,A -85,B 0,C 180,E1 -4057.508,E2 -4057.508} C_VEL
LIN {X 0,Y 537.972,Z 834.484,A -85,B 0,C 180,E1 -4058.64,E2 -4058.64} C_VEL
LIN {X 0,Y 538.142,Z 826.342,A -85,B 0,C 180,E1 -4059.584,E2 -4059.584} C_VEL
LIN {X 0,Y 538.374,Z 816.408,A -85,B 0,C 180,E1 -4060.53,E2 -4060.53} C_VEL
LIN {X 0,Y 538.564,Z 806.604,A -85,B 0,C 180,E1 -4061.287,E2 -4061.287} C_VEL
LIN {X 0,Y 538.803,Z 795.719,A -85,B 0,C 180,E1 -4061.963,E2 -4061.963} C_VEL
LIN {X 0,Y 538.962,Z 783.125,A -85,B 0,C 180,E1 -4062.567,E2 -4062.567} C_VEL
LIN {X 0,Y 539.181,Z 770.121,A -85,B 0,C 180,E1 -4063.017,E2 -4063.017} C_VEL
LIN {X 0,Y 539.341,Z 757.161,A -85,B 0,C 180,E1 -4063.3,E2 -4063.3} C_VEL
LIN {X 0,Y 539.585,Z 658.687,A -85,B 0,C 180,E1 -4064.625,E2 -4064.625} C_VEL
LIN {X 0,Y 538.454,Z 651.203,A -85,B 0,C 180,E1 -4064.779,E2 -4064.779} C_VEL
LIN {X 0,Y 538.82,Z 629.984,A -85,B 0,C 180,E1 -4067.793,E2 -4067.793} C_VEL
LIN {X 0,Y 539.215,Z 610.013,A -85,B 0,C 180,E1 -4070.603,E2 -4070.603} C_VEL
LIN {X 0,Y 539.641,Z 587.536,A -85,B 0,C 180,E1 -4073.81,E2 -4073.81} C_VEL
LIN {X 0,Y 538.773,Z 581.891,A -85,B 0,C 180,E1 -4074.671,E2 -4074.671} C_VEL
LIN {X 0,Y 538.1,Z 578.458,A -85,B 0,C 180,E1 -4075.22,E2 -4075.22} C_VEL
LIN {X 0,Y 538.045,Z 578.464,A -85,B 0,C 180,E1 -4078.048,E2 -4078.048} C_VEL
LIN {X 0,Y 538.018,Z 578.472,A -85,B 0,C 180,E1 -4080.626,E2 -4080.626} C_VEL
LIN {X 0,Y 538.043,Z 578.461,A -85,B 0,C 180,E1 -4083.282,E2 -4083.282} C_VEL
LIN {X 0,Y 538.025,Z 578.464,A -85,B 0,C 180,E1 -4086.001,E2 -4086.001} C_VEL
LIN {X 0,Y 538.012,Z 578.469,A -85,B 0,C 180,E1 -4088.829,E2 -4088.829} C_VEL
LIN {X 0,Y 538.074,Z 578.462,A -85,B 0,C 180,E1 -4090.772,E2 -4090.772} C_VEL
LIN {X 0,Y 538.025,Z 578.466,A -85,B 0,C 180,E1 -4094.074,E2 -4094.074} C_VEL
LIN {X 0,Y 538.019,Z 578.463,A -85,B 0,C 180,E1 -4097.214,E2 -4097.214} C_VEL
LIN {X 0,Y 538.053,Z 578.463,A -85,B 0,C 180,E1 -4100.205,E2 -4100.205} C_VEL
LIN {X 0,Y 538.024,Z 578.462,A -85,B 0,C 180,E1 -4103.067,E2 -4103.067} C_VEL
LIN {X 0,Y 538.026,Z 578.462,A -85,B 0,C 180,E1 -4105.827,E2 -4105.827} C_VEL
LIN {X 0,Y 538.019,Z 578.469,A -85,B 0,C 180,E1 -4108.499,E2 -4108.499} C_VEL
LIN {X 0,Y 538.053,Z 578.457,A -85,B 0,C 180,E1 -4111.099,E2 -4111.099} C_VEL
LIN {X 0,Y 538.044,Z 578.458,A -85,B 0,C 180,E1 -4113.633,E2 -4113.633} C_VEL
LIN {X 0,Y 538.015,Z 578.467,A -85,B 0,C 180,E1 -4116.117,E2 -4116.117} C_VEL
LIN {X 0,Y 538.032,Z 578.459,A -85,B 0,C 180,E1 -4119.348,E2 -4119.348} C_VEL
LIN {X 0,Y 538.065,Z 578.464,A -85,B 0,C 180,E1 -4122.517,E2 -4122.517} C_VEL
LIN {X 0,Y 538.056,Z 578.457,A -85,B 0,C 180,E1 -4125.63,E2 -4125.63} C_VEL
LIN {X 0,Y 538.069,Z 578.46,A -85,B 0,C 180,E1 -4128.701,E2 -4128.701} C_VEL
LIN {X 0,Y 538.083,Z 578.456,A -85,B 0,C 180,E1 -4131.739,E2 -4131.739} C_VEL
LIN {X 0,Y 538.158,Z 578.448,A -85,B 0,C 180,E1 -4134.755,E2 -4134.755} C_VEL
LIN {X 0,Y 538.16,Z 578.446,A -85,B 0,C 180,E1 -4137.755,E2 -4137.755} C_VEL
LIN {X 0,Y 538.177,Z 578.446,A -85,B 0,C 180,E1 -4140.748,E2 -4140.748} C_VEL
LIN {X 0,Y 538.135,Z 578.449,A -85,B 0,C 180,E1 -4142.994,E2 -4142.994} C_VEL
LIN {X 0,Y 538.126,Z 578.455,A -85,B 0,C 180,E1 -4145.997,E2 -4145.997} C_VEL
LIN {X 0,Y 538.07,Z 578.457,A -85,B 0,C 180,E1 -4149.018,E2 -4149.018} C_VEL
LIN {X 0,Y 538.076,Z 578.462,A -85,B 0,C 180,E1 -4152.063,E2 -4152.063} C_VEL
LIN {X 0,Y 538.038,Z 578.465,A -85,B 0,C 180,E1 -4155.144,E2 -4155.144} C_VEL
LIN {X 0,Y 538.137,Z 578.617,A -85,B 0,C 180,E1 -4157.088,E2 -4157.088} C_VEL
LIN {X 0,Y 538.249,Z 584.083,A -85,B 0,C 180,E1 -4158.262,E2 -4158.262} C_VEL
LIN {X 0,Y 538.044,Z 594.029,A -85,B 0,C 180,E1 -4160.314,E2 -4160.314} C_VEL
LIN {X 0,Y 539.681,Z 604.145,A -85,B 0,C 180,E1 -4160.496,E2 -4160.496} C_VEL
LIN {X 0,Y 539.297,Z 700.499,A -85,B 0,C 180,E1 -4161.802,E2 -4161.802} C_VEL
LIN {X 0,Y 539.123,Z 713.272,A -85,B 0,C 180,E1 -4162.129,E2 -4162.129} C_VEL
LIN {X 0,Y 538.93,Z 725.697,A -85,B 0,C 180,E1 -4162.585,E2 -4162.585} C_VEL
LIN {X 0,Y 538.76,Z 736.758,A -85,B 0,C 180,E1 -4163.14,E2 -4163.14} C_VEL
LIN {X 0,Y 538.636,Z 741.748,A -85,B 0,C 180,E1 -4163.437,E2 -4163.437} C_VEL
LIN {X 0,Y 537.908,Z 746.804,A -85,B 0,C 180,E1 -4163.759,E2 -4163.759} C_VEL
LIN {X 0,Y 534.884,Z 754.756,A -85,B 0,C 180,E1 -4164.306,E2 -4164.306} C_VEL
LIN {X 0,Y 531.836,Z 762.238,A -85,B 0,C 180,E1 -4164.923,E2 -4164.923} C_VEL
LIN {X 0,Y 531.076,Z 766.516,A -85,B 0,C 180,E1 -4165.351,E2 -4165.351} C_VEL
LIN {X 0,Y 530.843,Z 774.814,A -85,B 0,C 180,E1 -4166.328,E2 -4166.328} C_VEL
LIN {X 0,Y 530.711,Z 782.678,A -85,B 0,C 180,E1 -4167.472,E2 -4167.472} C_VEL
LIN {X 0,Y 530.594,Z 789.742,A -85,B 0,C 180,E1 -4168.76,E2 -4168.76} C_VEL
LIN {X 0,Y 530.502,Z 794.202,A -85,B 0,C 180,E1 -4169.788,E2 -4169.788} C_VEL
LIN {X 0,Y 530.462,Z 798.589,A -85,B 0,C 180,E1 -4171.111,E2 -4171.111} C_VEL
LIN {X 0,Y 530.407,Z 800.8,A -85,B 0,C 180,E1 -4172.006,E2 -4172.006} C_VEL
LIN {X 0,Y 530.353,Z 803.058,A -85,B 0,C 180,E1 -4173.402,E2 -4173.402} C_VEL
LIN {X 0,Y 530.369,Z 803.948,A -85,B 0,C 180,E1 -4174.76,E2 -4174.76} C_VEL
LIN {X 0,Y 530.334,Z 803.624,A -85,B 0,C 180,E1 -4176.065,E2 -4176.065} C_VEL
LIN {X 0,Y 530.351,Z 801.803,A -85,B 0,C 180,E1 -4177.559,E2 -4177.559} C_VEL
LIN {X 0,Y 530.428,Z 798.515,A -85,B 0,C 180,E1 -4179.006,E2 -4179.006} C_VEL
LIN {X 0,Y 530.501,Z 794.94,A -85,B 0,C 180,E1 -4180.103,E2 -4180.103} C_VEL
LIN {X 0,Y 530.54,Z 790.364,A -85,B 0,C 180,E1 -4181.197,E2 -4181.197} C_VEL
LIN {X 0,Y 530.678,Z 783.493,A -85,B 0,C 180,E1 -4182.486,E2 -4182.486} C_VEL
LIN {X 0,Y 530.833,Z 776.696,A -85,B 0,C 180,E1 -4183.508,E2 -4183.508} C_VEL
LIN {X 0,Y 531.06,Z 767.165,A -85,B 0,C 180,E1 -4184.672,E2 -4184.672} C_VEL
LIN {X 0,Y 531.3,Z 757.871,A -85,B 0,C 180,E1 -4185.587,E2 -4185.587} C_VEL
LIN {X 0,Y 531.545,Z 746.425,A -85,B 0,C 180,E1 -4186.494,E2 -4186.494} C_VEL
LIN {X 0,Y 531.825,Z 735.62,A -85,B 0,C 180,E1 -4187.174,E2 -4187.174} C_VEL
LIN {X 0,Y 532.07,Z 723.163,A -85,B 0,C 180,E1 -4187.776,E2 -4187.776} C_VEL
LIN {X 0,Y 532.257,Z 709.813,A -85,B 0,C 180,E1 -4188.244,E2 -4188.244} C_VEL
LIN {X 0,Y 532.442,Z 696.629,A -85,B 0,C 180,E1 -4188.53,E2 -4188.53} C_VEL
LIN {X 0,Y 532.707,Z 603.034,A -85,B 0,C 180,E1 -4189.804,E2 -4189.804} C_VEL
LIN {X 0,Y 531.065,Z 594.093,A -85,B 0,C 180,E1 -4189.986,E2 -4189.986} C_VEL
LIN {X 0,Y 531.34,Z 582.155,A -85,B 0,C 180,E1 -4192.525,E2 -4192.525} C_VEL
LIN {X 0,Y 531.053,Z 579.337,A -85,B 0,C 180,E1 -4193.155,E2 -4193.155} C_VEL
LIN {X 0,Y 530.997,Z 579.339,A -85,B 0,C 180,E1 -4196.495,E2 -4196.495} C_VEL
LIN {X 0,Y 530.97,Z 579.341,A -85,B 0,C 180,E1 -4199.356,E2 -4199.356} C_VEL
LIN {X 0,Y 531.014,Z 579.337,A -85,B 0,C 180,E1 -4202.468,E2 -4202.468} C_VEL
LIN {X 0,Y 531.004,Z 579.335,A -85,B 0,C 180,E1 -4204.943,E2 -4204.943} C_VEL
LIN {X 0,Y 530.97,Z 579.347,A -85,B 0,C 180,E1 -4208.248,E2 -4208.248} C_VEL
LIN {X 0,Y 530.995,Z 579.339,A -85,B 0,C 180,E1 -4210.678,E2 -4210.678} C_VEL
LIN {X 0,Y 530.992,Z 579.337,A -85,B 0,C 180,E1 -4213.072,E2 -4213.072} C_VEL
LIN {X 0,Y 531.02,Z 579.333,A -85,B 0,C 180,E1 -4215.437,E2 -4215.437} C_VEL
LIN {X 0,Y 531.049,Z 579.336,A -85,B 0,C 180,E1 -4218.551,E2 -4218.551} C_VEL
LIN {X 0,Y 531.056,Z 579.329,A -85,B 0,C 180,E1 -4221.63,E2 -4221.63} C_VEL
LIN {X 0,Y 531.121,Z 579.326,A -85,B 0,C 180,E1 -4224.686,E2 -4224.686} C_VEL
LIN {X 0,Y 531.142,Z 579.318,A -85,B 0,C 180,E1 -4227.726,E2 -4227.726} C_VEL
LIN {X 0,Y 531.155,Z 579.323,A -85,B 0,C 180,E1 -4230.759,E2 -4230.759} C_VEL
LIN {X 0,Y 531.109,Z 579.325,A -85,B 0,C 180,E1 -4233.035,E2 -4233.035} C_VEL
LIN {X 0,Y 531.086,Z 579.326,A -85,B 0,C 180,E1 -4236.078,E2 -4236.078} C_VEL
LIN {X 0,Y 531.034,Z 579.334,A -85,B 0,C 180,E1 -4239.139,E2 -4239.139} C_VEL
LIN {X 0,Y 531.045,Z 579.332,A -85,B 0,C 180,E1 -4242.226,E2 -4242.226} C_VEL
LIN {X 0,Y 530.999,Z 579.338,A -85,B 0,C 180,E1 -4245.35,E2 -4245.35} C_VEL
LIN {X 0,Y 530.992,Z 579.341,A -85,B 0,C 180,E1 -4248.522,E2 -4248.522} C_VEL
LIN {X 0,Y 531.003,Z 579.345,A -85,B 0,C 180,E1 -4250.939,E2 -4250.939} C_VEL
LIN {X 0,Y 530.975,Z 579.339,A -85,B 0,C 180,E1 -4254.225,E2 -4254.225} C_VEL
LIN {X 0,Y 531.009,Z 579.339,A -85,B 0,C 180,E1 -4256.744,E2 -4256.744} C_VEL
LIN {X 0,Y 530.986,Z 579.343,A -85,B 0,C 180,E1 -4259.323,E2 -4259.323} C_VEL
LIN {X 0,Y 530.969,Z 579.339,A -85,B 0,C 180,E1 -4262.101,E2 -4262.101} C_VEL
LIN {X 0,Y 530.984,Z 579.342,A -85,B 0,C 180,E1 -4264.853,E2 -4264.853} C_VEL
LIN {X 0,Y 530.97,Z 579.344,A -85,B 0,C 180,E1 -4267.508,E2 -4267.508} C_VEL
LIN {X 0,Y 530.986,Z 579.337,A -85,B 0,C 180,E1 -4270.433,E2 -4270.433} C_VEL
LIN {X 0,Y 530.965,Z 579.349,A -85,B 0,C 180,E1 -4273.281,E2 -4273.281} C_VEL
LIN {X 0,Y 530.986,Z 579.343,A -85,B 0,C 180,E1 -4275.622,E2 -4275.622} C_VEL
LIN {X 0,Y 531.001,Z 579.335,A -85,B 0,C 180,E1 -4278.565,E2 -4278.565} C_VEL
LIN {X 0,Y 530.963,Z 579.349,A -85,B 0,C 180,E1 -4281.53,E2 -4281.53} C_VEL
LIN {X 0,Y 530.959,Z 579.341,A -85,B 0,C 180,E1 -4284.38,E2 -4284.38} C_VEL
LIN {X 0,Y 530.972,Z 579.342,A -85,B 0,C 180,E1 -4287.134,E2 -4287.134} C_VEL
LIN {X 0,Y 530.974,Z 579.346,A -85,B 0,C 180,E1 -4289.803,E2 -4289.803} C_VEL
LIN {X 0,Y 531.017,Z 579.334,A -85,B 0,C 180,E1 -4292.468,E2 -4292.468} C_VEL
LIN {X 0,Y 530.999,Z 579.336,A -85,B 0,C 180,E1 -4294.942,E2 -4294.942} C_VEL
LIN {X 0,Y 530.976,Z 579.341,A -85,B 0,C 180,E1 -4298.247,E2 -4298.247} C_VEL
LIN {X 0,Y 530.997,Z 579.336,A -85,B 0,C 180,E1 -4300.677,E2 -4300.677} C_VEL
LIN {X 0,Y 530.98,Z 579.338,A -85,B 0,C 180,E1 -4303.071,E2 -4303.071} C_VEL
LIN {X 0,Y 531.024,Z 579.335,A -85,B 0,C 180,E1 -4305.436,E2 -4305.436} C_VEL
LIN {X 0,Y 531.042,Z 579.332,A -85,B 0,C 180,E1 -4308.55,E2 -4308.55} C_VEL
LIN {X 0,Y 531.057,Z 579.332,A -85,B 0,C 180,E1 -4311.63,E2 -4311.63} C_VEL
LIN {X 0,Y 531.126,Z 579.321,A -85,B 0,C 180,E1 -4314.685,E2 -4314.685} C_VEL
LIN {X 0,Y 531.145,Z 579.321,A -85,B 0,C 180,E1 -4317.725,E2 -4317.725} C_VEL
LIN {X 0,Y 531.158,Z 579.318,A -85,B 0,C 180,E1 -4320.758,E2 -4320.758} C_VEL
LIN {X 0,Y 531.11,Z 579.322,A -85,B 0,C 180,E1 -4323.034,E2 -4323.034} C_VEL
LIN {X 0,Y 531.086,Z 579.331,A -85,B 0,C 180,E1 -4326.077,E2 -4326.077} C_VEL
LIN {X 0,Y 531.058,Z 579.338,A -85,B 0,C 180,E1 -4328.371,E2 -4328.371} C_VEL
LIN {X 0,Y 531.057,Z 579.329,A -85,B 0,C 180,E1 -4331.672,E2 -4331.672} C_VEL
LIN {X 0,Y 531.037,Z 579.333,A -85,B 0,C 180,E1 -4334.956,E2 -4334.956} C_VEL
LIN {X 0,Y 530.987,Z 579.337,A -85,B 0,C 180,E1 -4337.724,E2 -4337.724} C_VEL
LIN {X 0,Y 531.03,Z 579.335,A -85,B 0,C 180,E1 -4340.127,E2 -4340.127} C_VEL
LIN {X 0,Y 530.951,Z 579.351,A -85,B 0,C 180,E1 -4342.573,E2 -4342.573} C_VEL
LIN {X 0,Y 531.01,Z 579.338,A -85,B 0,C 180,E1 -4345.057,E2 -4345.057} C_VEL
LIN {X 0,Y 531.018,Z 579.333,A -85,B 0,C 180,E1 -4347.596,E2 -4347.596} C_VEL
LIN {X 0,Y 530.98,Z 579.346,A -85,B 0,C 180,E1 -4350.645,E2 -4350.645} C_VEL
LIN {X 0,Y 530.994,Z 579.336,A -85,B 0,C 180,E1 -4353.772,E2 -4353.772} C_VEL
LIN {X 0,Y 530.96,Z 579.345,A -85,B 0,C 180,E1 -4356.558,E2 -4356.558} C_VEL
LIN {X 0,Y 530.992,Z 579.339,A -85,B 0,C 180,E1 -4359.443,E2 -4359.443} C_VEL
LIN {X 0,Y 530.985,Z 579.34,A -85,B 0,C 180,E1 -4362.456,E2 -4362.456} C_VEL
LIN {X 0,Y 530.988,Z 579.338,A -85,B 0,C 180,E1 -4365.621,E2 -4365.621} C_VEL
LIN {X 0,Y 530.999,Z 579.338,A -85,B 0,C 180,E1 -4368.564,E2 -4368.564} C_VEL
LIN {X 0,Y 530.963,Z 579.344,A -85,B 0,C 180,E1 -4371.529,E2 -4371.529} C_VEL
LIN {X 0,Y 530.962,Z 579.34,A -85,B 0,C 180,E1 -4374.38,E2 -4374.38} C_VEL
LIN {X 0,Y 530.976,Z 579.348,A -85,B 0,C 180,E1 -4377.133,E2 -4377.133} C_VEL
LIN {X 0,Y 530.967,Z 579.344,A -85,B 0,C 180,E1 -4379.802,E2 -4379.802} C_VEL
LIN {X 0,Y 531.018,Z 579.336,A -85,B 0,C 180,E1 -4382.467,E2 -4382.467} C_VEL
LIN {X 0,Y 531.068,Z 579.487,A -85,B 0,C 180,E1 -4384.578,E2 -4384.578} C_VEL
LIN {X 0,Y 532.766,Z 589,A -85,B 0,C 180,E1 -4386.068,E2 -4386.068} C_VEL
LIN {X 0,Y 532.357,Z 607.108,A -85,B 0,C 180,E1 -4388.712,E2 -4388.712} C_VEL
LIN {X 0,Y 531.888,Z 628.952,A -85,B 0,C 180,E1 -4391.858,E2 -4391.858} C_VEL
LIN {X 0,Y 531.447,Z 651.359,A -85,B 0,C 180,E1 -4395.045,E2 -4395.045} C_VEL
LIN {X 0,Y 532.842,Z 661.343,A -85,B 0,C 180,E1 -4395.222,E2 -4395.222} C_VEL
LIN {X 0,Y 532.439,Z 759.91,A -85,B 0,C 180,E1 -4396.571,E2 -4396.571} C_VEL
LIN {X 0,Y 532.257,Z 773.193,A -85,B 0,C 180,E1 -4396.906,E2 -4396.906} C_VEL
LIN {X 0,Y 532.005,Z 786.471,A -85,B 0,C 180,E1 -4397.409,E2 -4397.409} C_VEL
LIN {X 0,Y 531.802,Z 797.964,A -85,B 0,C 180,E1 -4398.007,E2 -4398.007} C_VEL
LIN {X 0,Y 531.529,Z 809.183,A -85,B 0,C 180,E1 -4398.753,E2 -4398.753} C_VEL
LIN {X 0,Y 531.256,Z 819.597,A -85,B 0,C 180,E1 -4399.615,E2 -4399.615} C_VEL
LIN {X 0,Y 531.061,Z 828.106,A -85,B 0,C 180,E1 -4400.477,E2 -4400.477} C_VEL
LIN {X 0,Y 530.885,Z 835.955,A -85,B 0,C 180,E1 -4401.434,E2 -4401.434} C_VEL
LIN {X 0,Y 530.686,Z 843.617,A -85,B 0,C 180,E1 -4402.58,E2 -4402.58} C_VEL
LIN {X 0,Y 530.605,Z 850.676,A -85,B 0,C 180,E1 -4403.917,E2 -4403.917} C_VEL
LIN {X 0,Y 530.459,Z 855.37,A -85,B 0,C 180,E1 -4405.059,E2 -4405.059} C_VEL
LIN {X 0,Y 530.516,Z 858.956,A -85,B 0,C 180,E1 -4406.201,E2 -4406.201} C_VEL
LIN {X 0,Y 530.457,Z 860.805,A -85,B 0,C 180,E1 -4406.961,E2 -4406.961} C_VEL
LIN {X 0,Y 530.41,Z 862.193,A -85,B 0,C 180,E1 -4407.721,E2 -4407.721} C_VEL
LIN {X 0,Y 530.344,Z 863.785,A -85,B 0,C 180,E1 -4409.24,E2 -4409.24} C_VEL
LIN {X 0,Y 530.342,Z 864,A -85,B 0,C 180,E1 -4409.999,E2 -4409.999} C_VEL
LIN {X 0,Y 530.361,Z 863.185,A -85,B 0,C 180,E1 -4411.518,E2 -4411.518} C_VEL
LIN {X 0,Y 530.41,Z 862.198,A -85,B 0,C 180,E1 -4412.277,E2 -4412.277} C_VEL
LIN {X 0,Y 530.457,Z 860.812,A -85,B 0,C 180,E1 -4413.037,E2 -4413.037} C_VEL
LIN {X 0,Y 530.522,Z 857.898,A -85,B 0,C 180,E1 -4414.177,E2 -4414.177} C_VEL
LIN {X 0,Y 530.524,Z 853.951,A -85,B 0,C 180,E1 -4415.32,E2 -4415.32} C_VEL
LIN {X 0,Y 530.595,Z 848.283,A -85,B 0,C 180,E1 -4416.578,E2 -4416.578} C_VEL
LIN {X 0,Y 530.757,Z 841.241,A -85,B 0,C 180,E1 -4417.8,E2 -4417.8} C_VEL
LIN {X 0,Y 530.929,Z 832.999,A -85,B 0,C 180,E1 -4418.947,E2 -4418.947} C_VEL
LIN {X 0,Y 531.136,Z 824.548,A -85,B 0,C 180,E1 -4419.904,E2 -4419.904} C_VEL
LIN {X 0,Y 531.408,Z 814.103,A -85,B 0,C 180,E1 -4420.862,E2 -4420.862} C_VEL
LIN {X 0,Y 531.702,Z 803.149,A -85,B 0,C 180,E1 -4421.67,E2 -4421.67} C_VEL
LIN {X 0,Y 531.93,Z 792.421,A -85,B 0,C 180,E1 -4422.3,E2 -4422.3} C_VEL
LIN {X 0,Y 532.139,Z 780.788,A -85,B 0,C 180,E1 -4422.828,E2 -4422.828} C_VEL
LIN {X 0,Y 532.289,Z 767.379,A -85,B 0,C 180,E1 -4423.261,E2 -4423.261} C_VEL
LIN {X 0,Y 532.454,Z 754.146,A -85,B 0,C 180,E1 -4423.524,E2 -4423.524} C_VEL
LIN {X 0,Y 532.684,Z 659.106,A -85,B 0,C 180,E1 -4424.813,E2 -4424.813} C_VEL
LIN {X 0,Y 531.476,Z 651.355,A -85,B 0,C 180,E1 -4424.955,E2 -4424.955} C_VEL
LIN {X 0,Y 531.853,Z 628.791,A -85,B 0,C 180,E1 -4428.144,E2 -4428.144} C_VEL
LIN {X 0,Y 532.306,Z 606.775,A -85,B 0,C 180,E1 -4431.288,E2 -4431.288} C_VEL
LIN {X 0,Y 532.696,Z 588.527,A -85,B 0,C 180,E1 -4433.934,E2 -4433.934} C_VEL
LIN {X 0,Y 531.03,Z 579.338,A -85,B 0,C 180,E1 -4435.396,E2 -4435.396} C_VEL
LIN {X 0,Y 530.998,Z 579.345,A -85,B 0,C 180,E1 -4438.454,E2 -4438.454} C_VEL
LIN {X 0,Y 530.955,Z 579.347,A -85,B 0,C 180,E1 -4441.078,E2 -4441.078} C_VEL
LIN {X 0,Y 530.988,Z 579.34,A -85,B 0,C 180,E1 -4443.771,E2 -4443.771} C_VEL
LIN {X 0,Y 530.966,Z 579.35,A -85,B 0,C 180,E1 -4446.556,E2 -4446.556} C_VEL
LIN {X 0,Y 531.003,Z 579.339,A -85,B 0,C 180,E1 -4449.856,E2 -4449.856} C_VEL
LIN {X 0,Y 530.976,Z 579.349,A -85,B 0,C 180,E1 -4452.455,E2 -4452.455} C_VEL
LIN {X 0,Y 530.983,Z 579.34,A -85,B 0,C 180,E1 -4455.62,E2 -4455.62} C_VEL
LIN {X 0,Y 531.002,Z 579.344,A -85,B 0,C 180,E1 -4458.565,E2 -4458.565} C_VEL
LIN {X 0,Y 530.966,Z 579.34,A -85,B 0,C 180,E1 -4461.345,E2 -4461.345} C_VEL
LIN {X 0,Y 530.977,Z 579.346,A -85,B 0,C 180,E1 -4464.381,E2 -4464.381} C_VEL
LIN {X 0,Y 530.969,Z 579.341,A -85,B 0,C 180,E1 -4467.133,E2 -4467.133} C_VEL
LIN {X 0,Y 530.98,Z 579.339,A -85,B 0,C 180,E1 -4469.803,E2 -4469.803} C_VEL
LIN {X 0,Y 531.011,Z 579.343,A -85,B 0,C 180,E1 -4472.466,E2 -4472.466} C_VEL
LIN {X 0,Y 531.001,Z 579.338,A -85,B 0,C 180,E1 -4474.942,E2 -4474.942} C_VEL
LIN {X 0,Y 530.964,Z 579.347,A -85,B 0,C 180,E1 -4478.246,E2 -4478.246} C_VEL
LIN {X 0,Y 530.99,Z 579.343,A -85,B 0,C 180,E1 -4480.677,E2 -4480.677} C_VEL
LIN {X 0,Y 530.984,Z 579.339,A -85,B 0,C 180,E1 -4483.071,E2 -4483.071} C_VEL
LIN {X 0,Y 531.011,Z 579.334,A -85,B 0,C 180,E1 -4485.435,E2 -4485.435} C_VEL
LIN {X 0,Y 531.041,Z 579.338,A -85,B 0,C 180,E1 -4488.55,E2 -4488.55} C_VEL
LIN {X 0,Y 531.052,Z 579.331,A -85,B 0,C 180,E1 -4491.629,E2 -4491.629} C_VEL
LIN {X 0,Y 531.116,Z 579.326,A -85,B 0,C 180,E1 -4494.685,E2 -4494.685} C_VEL
LIN {X 0,Y 531.132,Z 579.322,A -85,B 0,C 180,E1 -4497.725,E2 -4497.725} C_VEL
LIN {X 0,Y 531.147,Z 579.322,A -85,B 0,C 180,E1 -4500.758,E2 -4500.758} C_VEL
LIN {X 0,Y 531.102,Z 579.325,A -85,B 0,C 180,E1 -4503.034,E2 -4503.034} C_VEL
LIN {X 0,Y 531.084,Z 579.334,A -85,B 0,C 180,E1 -4506.077,E2 -4506.077} C_VEL
LIN {X 0,Y 531.029,Z 579.334,A -85,B 0,C 180,E1 -4509.138,E2 -4509.138} C_VEL
LIN {X 0,Y 531.033,Z 579.342,A -85,B 0,C 180,E1 -4512.225,E2 -4512.225} C_VEL
LIN {X 0,Y 530.99,Z 579.343,A -85,B 0,C 180,E1 -4515.35,E2 -4515.35} C_VEL
LIN {X 0,Y 531.073,Z 579.435,A -85,B 0,C 180,E1 -4516.926,E2 -4516.926} C_VEL
LIN {X 0,Y 531.329,Z 583.224,A -85,B 0,C 180,E1 -4517.761,E2 -4517.761} C_VEL
LIN {X 0,Y 531.04,Z 594.204,A -85,B 0,C 180,E1 -4520.112,E2 -4520.112} C_VEL
LIN {X 0,Y 532.816,Z 604.394,A -85,B 0,C 180,E1 -4520.307,E2 -4520.307} C_VEL
LIN {X 0,Y 532.412,Z 699.895,A -85,B 0,C 180,E1 -4521.615,E2 -4521.615} C_VEL
LIN {X 0,Y 532.199,Z 712.547,A -85,B 0,C 180,E1 -4521.934,E2 -4521.934} C_VEL
LIN {X 0,Y 532.03,Z 724.814,A -85,B 0,C 180,E1 -4522.382,E2 -4522.382} C_VEL
LIN {X 0,Y 531.818,Z 736.129,A -85,B 0,C 180,E1 -4522.945,E2 -4522.945} C_VEL
LIN {X 0,Y 531.569,Z 747.547,A -85,B 0,C 180,E1 -4523.678,E2 -4523.678} C_VEL
LIN {X 0,Y 531.27,Z 758.093,A -85,B 0,C 180,E1 -4524.522,E2 -4524.522} C_VEL
LIN {X 0,Y 531.076,Z 766.516,A -85,B 0,C 180,E1 -4525.351,E2 -4525.351} C_VEL
LIN {X 0,Y 530.324,Z 770.667,A -85,B 0,C 180,E1 -4525.803,E2 -4525.803} C_VEL
LIN {X 0,Y 525.954,Z 779.344,A -85,B 0,C 180,E1 -4526.882,E2 -4526.882} C_VEL
LIN {X 0,Y 523.934,Z 783.818,A -85,B 0,C 180,E1 -4527.561,E2 -4527.561} C_VEL
LIN {X 0,Y 523.608,Z 785.881,A -85,B 0,C 180,E1 -4527.924,E2 -4527.924} C_VEL
LIN {X 0,Y 523.463,Z 792.237,A -85,B 0,C 180,E1 -4529.23,E2 -4529.23} C_VEL
LIN {X 0,Y 523.387,Z 797.491,A -85,B 0,C 180,E1 -4530.681,E2 -4530.681} C_VEL
LIN {X 0,Y 523.337,Z 799.943,A -85,B 0,C 180,E1 -4531.583,E2 -4531.583} C_VEL
LIN {X 0,Y 523.272,Z 801.804,A -85,B 0,C 180,E1 -4532.496,E2 -4532.496} C_VEL
LIN {X 0,Y 523.273,Z 803.304,A -85,B 0,C 180,E1 -4533.624,E2 -4533.624} C_VEL
LIN {X 0,Y 523.267,Z 803.995,A -85,B 0,C 180,E1 -4534.988,E2 -4534.988} C_VEL
LIN {X 0,Y 523.24,Z 803.465,A -85,B 0,C 180,E1 -4536.305,E2 -4536.305} C_VEL
LIN {X 0,Y 523.251,Z 801.81,A -85,B 0,C 180,E1 -4537.587,E2 -4537.587} C_VEL
LIN {X 0,Y 523.356,Z 798.312,A -85,B 0,C 180,E1 -4539.135,E2 -4539.135} C_VEL
LIN {X 0,Y 523.453,Z 793.169,A -85,B 0,C 180,E1 -4540.63,E2 -4540.63} C_VEL
LIN {X 0,Y 523.522,Z 787.243,A -85,B 0,C 180,E1 -4541.917,E2 -4541.917} C_VEL
LIN {X 0,Y 523.691,Z 779.692,A -85,B 0,C 180,E1 -4543.19,E2 -4543.19} C_VEL
LIN {X 0,Y 523.887,Z 772.084,A -85,B 0,C 180,E1 -4544.234,E2 -4544.234} C_VEL
LIN {X 0,Y 524.164,Z 762.671,A -85,B 0,C 180,E1 -4545.286,E2 -4545.286} C_VEL
LIN {X 0,Y 524.454,Z 752.513,A -85,B 0,C 180,E1 -4546.197,E2 -4546.197} C_VEL
LIN {X 0,Y 524.714,Z 741.797,A -85,B 0,C 180,E1 -4546.974,E2 -4546.974} C_VEL
LIN {X 0,Y 525.037,Z 729.676,A -85,B 0,C 180,E1 -4547.659,E2 -4547.659} C_VEL
LIN {X 0,Y 525.288,Z 718.082,A -85,B 0,C 180,E1 -4548.152,E2 -4548.152} C_VEL
LIN {X 0,Y 525.443,Z 705.745,A -85,B 0,C 180,E1 -4548.529,E2 -4548.529} C_VEL
LIN {X 0,Y 525.578,Z 691.499,A -85,B 0,C 180,E1 -4548.784,E2 -4548.784} C_VEL
LIN {X 0,Y 525.832,Z 604.05,A -85,B 0,C 180,E1 -4549.988,E2 -4549.988} C_VEL
LIN {X 0,Y 524.09,Z 594.432,A -85,B 0,C 180,E1 -4550.185,E2 -4550.185} C_VEL
LIN {X 0,Y 524.348,Z 583.245,A -85,B 0,C 180,E1 -4552.582,E2 -4552.582} C_VEL
LIN {X 0,Y 523.994,Z 580.217,A -85,B 0,C 180,E1 -4553.267,E2 -4553.267} C_VEL
LIN {X 0,Y 523.94,Z 580.217,A -85,B 0,C 180,E1 -4556.637,E2 -4556.637} C_VEL
LIN {X 0,Y 523.952,Z 580.215,A -85,B 0,C 180,E1 -4559.357,E2 -4559.357} C_VEL
LIN {X 0,Y 523.977,Z 580.216,A -85,B 0,C 180,E1 -4562.282,E2 -4562.282} C_VEL
LIN {X 0,Y 523.951,Z 580.216,A -85,B 0,C 180,E1 -4564.582,E2 -4564.582} C_VEL
LIN {X 0,Y 523.915,Z 580.218,A -85,B 0,C 180,E1 -4567.108,E2 -4567.108} C_VEL
LIN {X 0,Y 523.978,Z 580.215,A -85,B 0,C 180,E1 -4569.867,E2 -4569.867} C_VEL
LIN {X 0,Y 523.97,Z 580.213,A -85,B 0,C 180,E1 -4572.838,E2 -4572.838} C_VEL
LIN {X 0,Y 523.977,Z 580.21,A -85,B 0,C 180,E1 -4575.237,E2 -4575.237} C_VEL
LIN {X 0,Y 524.015,Z 580.214,A -85,B 0,C 180,E1 -4578.395,E2 -4578.395} C_VEL
LIN {X 0,Y 524.005,Z 580.207,A -85,B 0,C 180,E1 -4581.517,E2 -4581.517} C_VEL
LIN {X 0,Y 524.082,Z 580.204,A -85,B 0,C 180,E1 -4584.615,E2 -4584.615} C_VEL
LIN {X 0,Y 524.114,Z 580.193,A -85,B 0,C 180,E1 -4587.695,E2 -4587.695} C_VEL
LIN {X 0,Y 524.125,Z 580.198,A -85,B 0,C 180,E1 -4590.769,E2 -4590.769} C_VEL
LIN {X 0,Y 524.076,Z 580.201,A -85,B 0,C 180,E1 -4593.076,E2 -4593.076} C_VEL
LIN {X 0,Y 524.048,Z 580.204,A -85,B 0,C 180,E1 -4596.16,E2 -4596.16} C_VEL
LIN {X 0,Y 524.002,Z 580.209,A -85,B 0,C 180,E1 -4599.263,E2 -4599.263} C_VEL
LIN {X 0,Y 524.006,Z 580.207,A -85,B 0,C 180,E1 -4601.74,E2 -4601.74} C_VEL
LIN {X 0,Y 523.997,Z 580.214,A -85,B 0,C 180,E1 -4605.053,E2 -4605.053} C_VEL
LIN {X 0,Y 523.967,Z 580.211,A -85,B 0,C 180,E1 -4607.97,E2 -4607.97} C_VEL
LIN {X 0,Y 523.975,Z 580.213,A -85,B 0,C 180,E1 -4610.411,E2 -4610.411} C_VEL
LIN {X 0,Y 523.914,Z 580.227,A -85,B 0,C 180,E1 -4612.894,E2 -4612.894} C_VEL
LIN {X 0,Y 523.956,Z 580.216,A -85,B 0,C 180,E1 -4615.419,E2 -4615.419} C_VEL
LIN {X 0,Y 523.974,Z 580.211,A -85,B 0,C 180,E1 -4617.999,E2 -4617.999} C_VEL
LIN {X 0,Y 523.948,Z 580.219,A -85,B 0,C 180,E1 -4620.855,E2 -4620.855} C_VEL
LIN {X 0,Y 523.965,Z 580.214,A -85,B 0,C 180,E1 -4623.735,E2 -4623.735} C_VEL
LIN {X 0,Y 523.908,Z 580.219,A -85,B 0,C 180,E1 -4626.402,E2 -4626.402} C_VEL
LIN {X 0,Y 523.927,Z 580.223,A -85,B 0,C 180,E1 -4629.085,E2 -4629.085} C_VEL
LIN {X 0,Y 523.955,Z 580.213,A -85,B 0,C 180,E1 -4632.119,E2 -4632.119} C_VEL
LIN {X 0,Y 523.95,Z 580.223,A -85,B 0,C 180,E1 -4635.31,E2 -4635.31} C_VEL
LIN {X 0,Y 523.963,Z 580.213,A -85,B 0,C 180,E1 -4638.69,E2 -4638.69} C_VEL
LIN {X 0,Y 523.922,Z 580.221,A -85,B 0,C 180,E1 -4641.081,E2 -4641.081} C_VEL
LIN {X 0,Y 523.905,Z 580.224,A -85,B 0,C 180,E1 -4643.826,E2 -4643.826} C_VEL
LIN {X 0,Y 523.946,Z 580.214,A -85,B 0,C 180,E1 -4646.636,E2 -4646.636} C_VEL
LIN {X 0,Y 523.96,Z 580.218,A -85,B 0,C 180,E1 -4649.356,E2 -4649.356} C_VEL
LIN {X 0,Y 523.982,Z 580.211,A -85,B 0,C 180,E1 -4652.282,E2 -4652.282} C_VEL
LIN {X 0,Y 523.952,Z 580.214,A -85,B 0,C 180,E1 -4654.581,E2 -4654.581} C_VEL
LIN {X 0,Y 523.924,Z 580.227,A -85,B 0,C 180,E1 -4657.757,E2 -4657.757} C_VEL
LIN {X 0,Y 523.978,Z 580.212,A -85,B 0,C 180,E1 -4660.408,E2 -4660.408} C_VEL
LIN {X 0,Y 523.962,Z 580.212,A -85,B 0,C 180,E1 -4662.837,E2 -4662.837} C_VEL
LIN {X 0,Y 523.982,Z 580.211,A -85,B 0,C 180,E1 -4665.236,E2 -4665.236} C_VEL
LIN {X 0,Y 524.018,Z 580.209,A -85,B 0,C 180,E1 -4668.394,E2 -4668.394} C_VEL
LIN {X 0,Y 524.005,Z 580.209,A -85,B 0,C 180,E1 -4671.516,E2 -4671.516} C_VEL
LIN {X 0,Y 524.087,Z 580.199,A -85,B 0,C 180,E1 -4674.614,E2 -4674.614} C_VEL
LIN {X 0,Y 524.117,Z 580.196,A -85,B 0,C 180,E1 -4677.695,E2 -4677.695} C_VEL
LIN {X 0,Y 524.128,Z 580.193,A -85,B 0,C 180,E1 -4680.768,E2 -4680.768} C_VEL
LIN {X 0,Y 524.076,Z 580.198,A -85,B 0,C 180,E1 -4683.075,E2 -4683.075} C_VEL
LIN {X 0,Y 524.049,Z 580.209,A -85,B 0,C 180,E1 -4686.159,E2 -4686.159} C_VEL
LIN {X 0,Y 524.006,Z 580.214,A -85,B 0,C 180,E1 -4688.484,E2 -4688.484} C_VEL
LIN {X 0,Y 524.008,Z 580.207,A -85,B 0,C 180,E1 -4691.739,E2 -4691.739} C_VEL
LIN {X 0,Y 523.999,Z 580.209,A -85,B 0,C 180,E1 -4695.052,E2 -4695.052} C_VEL
LIN {X 0,Y 523.953,Z 580.215,A -85,B 0,C 180,E1 -4697.97,E2 -4697.97} C_VEL
LIN {X 0,Y 523.978,Z 580.217,A -85,B 0,C 180,E1 -4700.41,E2 -4700.41} C_VEL
LIN {X 0,Y 523.916,Z 580.223,A -85,B 0,C 180,E1 -4702.893,E2 -4702.893} C_VEL
LIN {X 0,Y 523.958,Z 580.213,A -85,B 0,C 180,E1 -4705.419,E2 -4705.419} C_VEL
LIN {X 0,Y 523.973,Z 580.212,A -85,B 0,C 180,E1 -4707.999,E2 -4707.999} C_VEL
LIN {X 0,Y 523.95,Z 580.222,A -85,B 0,C 180,E1 -4710.855,E2 -4710.855} C_VEL
LIN {X 0,Y 523.966,Z 580.212,A -85,B 0,C 180,E1 -4713.734,E2 -4713.734} C_VEL
LIN {X 0,Y 523.909,Z 580.222,A -85,B 0,C 180,E1 -4716.401,E2 -4716.401} C_VEL
LIN {X 0,Y 523.926,Z 580.223,A -85,B 0,C 180,E1 -4719.085,E2 -4719.085} C_VEL
LIN {X 0,Y 523.96,Z 580.213,A -85,B 0,C 180,E1 -4722.118,E2 -4722.118} C_VEL
LIN {X 0,Y 523.958,Z 580.218,A -85,B 0,C 180,E1 -4725.309,E2 -4725.309} C_VEL
LIN {X 0,Y 523.961,Z 580.216,A -85,B 0,C 180,E1 -4728.689,E2 -4728.689} C_VEL
LIN {X 0,Y 523.924,Z 580.226,A -85,B 0,C 180,E1 -4731.08,E2 -4731.08} C_VEL
LIN {X 0,Y 523.906,Z 580.22,A -85,B 0,C 180,E1 -4733.825,E2 -4733.825} C_VEL
LIN {X 0,Y 523.948,Z 580.217,A -85,B 0,C 180,E1 -4736.635,E2 -4736.635} C_VEL
LIN {X 0,Y 523.954,Z 580.222,A -85,B 0,C 180,E1 -4739.355,E2 -4739.355} C_VEL
LIN {X 0,Y 523.982,Z 580.213,A -85,B 0,C 180,E1 -4742.281,E2 -4742.281} C_VEL
LIN {X 0,Y 523.997,Z 580.312,A -85,B 0,C 180,E1 -4744.382,E2 -4744.382} C_VEL
LIN {X 0,Y 525.818,Z 590.049,A -85,B 0,C 180,E1 -4745.941,E2 -4745.941} C_VEL
LIN {X 0,Y 525.395,Z 608.159,A -85,B 0,C 180,E1 -4748.622,E2 -4748.622} C_VEL
LIN {X 0,Y 524.9,Z 629.264,A -85,B 0,C 180,E1 -4751.7,E2 -4751.7} C_VEL
LIN {X 0,Y 524.432,Z 651.011,A -85,B 0,C 180,E1 -4754.834,E2 -4754.834} C_VEL
LIN {X 0,Y 525.965,Z 661.849,A -85,B 0,C 180,E1 -4755.038,E2 -4755.038} C_VEL
LIN {X 0,Y 525.547,Z 759.633,A -85,B 0,C 180,E1 -4756.391,E2 -4756.391} C_VEL
LIN {X 0,Y 525.336,Z 773.009,A -85,B 0,C 180,E1 -4756.731,E2 -4756.731} C_VEL
LIN {X 0,Y 525.062,Z 786.373,A -85,B 0,C 180,E1 -4757.24,E2 -4757.24} C_VEL
LIN {X 0,Y 524.818,Z 798.898,A -85,B 0,C 180,E1 -4757.904,E2 -4757.904} C_VEL
LIN {X 0,Y 524.508,Z 810.473,A -85,B 0,C 180,E1 -4758.698,E2 -4758.698} C_VEL
LIN {X 0,Y 524.235,Z 820.638,A -85,B 0,C 180,E1 -4759.572,E2 -4759.572} C_VEL
LIN {X 0,Y 523.976,Z 829.779,A -85,B 0,C 180,E1 -4760.542,E2 -4760.542} C_VEL
LIN {X 0,Y 523.759,Z 838.682,A -85,B 0,C 180,E1 -4761.706,E2 -4761.706} C_VEL
LIN {X 0,Y 523.584,Z 845.844,A -85,B 0,C 180,E1 -4762.867,E2 -4762.867} C_VEL
LIN {X 0,Y 523.544,Z 852.363,A -85,B 0,C 180,E1 -4764.221,E2 -4764.221} C_VEL
LIN {X 0,Y 523.361,Z 856.674,A -85,B 0,C 180,E1 -4765.378,E2 -4765.378} C_VEL
LIN {X 0,Y 523.444,Z 858.956,A -85,B 0,C 180,E1 -4766.15,E2 -4766.15} C_VEL
LIN {X 0,Y 523.368,Z 860.805,A -85,B 0,C 180,E1 -4766.92,E2 -4766.92} C_VEL
LIN {X 0,Y 523.334,Z 862.192,A -85,B 0,C 180,E1 -4767.69,E2 -4767.69} C_VEL
LIN {X 0,Y 523.25,Z 863.785,A -85,B 0,C 180,E1 -4769.23,E2 -4769.23} C_VEL
LIN {X 0,Y 523.246,Z 864,A -85,B 0,C 180,E1 -4769.999,E2 -4769.999} C_VEL
LIN {X 0,Y 523.274,Z 863.184,A -85,B 0,C 180,E1 -4771.538,E2 -4771.538} C_VEL
LIN {X 0,Y 523.334,Z 862.197,A -85,B 0,C 180,E1 -4772.308,E2 -4772.308} C_VEL
LIN {X 0,Y 523.367,Z 860.812,A -85,B 0,C 180,E1 -4773.078,E2 -4773.078} C_VEL
LIN {X 0,Y 523.441,Z 857.898,A -85,B 0,C 180,E1 -4774.234,E2 -4774.234} C_VEL
LIN {X 0,Y 523.464,Z 853.951,A -85,B 0,C 180,E1 -4775.392,E2 -4775.392} C_VEL
LIN {X 0,Y 523.519,Z 848.746,A -85,B 0,C 180,E1 -4776.577,E2 -4776.577} C_VEL
LIN {X 0,Y 523.664,Z 842.472,A -85,B 0,C 180,E1 -4777.712,E2 -4777.712} C_VEL
LIN {X 0,Y 523.856,Z 834.484,A -85,B 0,C 180,E1 -4778.874,E2 -4778.874} C_VEL
LIN {X 0,Y 524.107,Z 826.341,A -85,B 0,C 180,E1 -4779.843,E2 -4779.843} C_VEL
LIN {X 0,Y 524.365,Z 816.406,A -85,B 0,C 180,E1 -4780.814,E2 -4780.814} C_VEL
LIN {X 0,Y 524.692,Z 805.096,A -85,B 0,C 180,E1 -4781.694,E2 -4781.694} C_VEL
LIN {X 0,Y 524.921,Z 794.142,A -85,B 0,C 180,E1 -4782.369,E2 -4782.369} C_VEL
LIN {X 0,Y 525.174,Z 781.854,A -85,B 0,C 180,E1 -4782.952,E2 -4782.952} C_VEL
LIN {X 0,Y 525.324,Z 768.949,A -85,B 0,C 180,E1 -4783.391,E2 -4783.391} C_VEL
LIN {X 0,Y 525.569,Z 755.27,A -85,B 0,C 180,E1 -4783.68,E2 -4783.68} C_VEL
LIN {X 0,Y 525.838,Z 660.123,A -85,B 0,C 180,E1 -4784.987,E2 -4784.987} C_VEL
LIN {X 0,Y 524.409,Z 650.963,A -85,B 0,C 180,E1 -4785.158,E2 -4785.158} C_VEL
LIN {X 0,Y 524.809,Z 630.778,A -85,B 0,C 180,E1 -4788.047,E2 -4788.047} C_VEL
LIN {X 0,Y 525.257,Z 610.518,A -85,B 0,C 180,E1 -4790.976,E2 -4790.976} C_VEL
LIN {X 0,Y 525.753,Z 590.924,A -85,B 0,C 180,E1 -4793.85,E2 -4793.85} C_VEL
LIN {X 0,Y 525.294,Z 586.568,A -85,B 0,C 180,E1 -4794.524,E2 -4794.524} C_VEL
LIN {X 0,Y 524.009,Z 580.213,A -85,B 0,C 180,E1 -4795.549,E2 -4795.549} C_VEL
LIN {X 0,Y 523.969,Z 580.217,A -85,B 0,C 180,E1 -4797.998,E2 -4797.998} C_VEL
LIN {X 0,Y 523.942,Z 580.223,A -85,B 0,C 180,E1 -4800.854,E2 -4800.854} C_VEL
LIN {X 0,Y 523.959,Z 580.216,A -85,B 0,C 180,E1 -4803.734,E2 -4803.734} C_VEL
LIN {X 0,Y 523.92,Z 580.226,A -85,B 0,C 180,E1 -4806.403,E2 -4806.403} C_VEL
LIN {X 0,Y 523.928,Z 580.221,A -85,B 0,C 180,E1 -4809.083,E2 -4809.083} C_VEL
LIN {X 0,Y 523.969,Z 580.214,A -85,B 0,C 180,E1 -4811.311,E2 -4811.311} C_VEL
LIN {X 0,Y 523.951,Z 580.222,A -85,B 0,C 180,E1 -4814.69,E2 -4814.69} C_VEL
LIN {X 0,Y 523.953,Z 580.217,A -85,B 0,C 180,E1 -4817.881,E2 -4817.881} C_VEL
LIN {X 0,Y 523.961,Z 580.216,A -85,B 0,C 180,E1 -4820.919,E2 -4820.919} C_VEL
LIN {X 0,Y 523.922,Z 580.218,A -85,B 0,C 180,E1 -4823.827,E2 -4823.827} C_VEL
LIN {X 0,Y 523.938,Z 580.222,A -85,B 0,C 180,E1 -4826.635,E2 -4826.635} C_VEL
LIN {X 0,Y 523.957,Z 580.213,A -85,B 0,C 180,E1 -4829.356,E2 -4829.356} C_VEL
LIN {X 0,Y 523.973,Z 580.217,A -85,B 0,C 180,E1 -4832.28,E2 -4832.28} C_VEL
LIN {X 0,Y 523.949,Z 580.221,A -85,B 0,C 180,E1 -4834.581,E2 -4834.581} C_VEL
LIN {X 0,Y 523.909,Z 580.22,A -85,B 0,C 180,E1 -4837.106,E2 -4837.106} C_VEL
LIN {X 0,Y 523.971,Z 580.213,A -85,B 0,C 180,E1 -4839.865,E2 -4839.865} C_VEL
LIN {X 0,Y 523.962,Z 580.216,A -85,B 0,C 180,E1 -4842.837,E2 -4842.837} C_VEL
LIN {X 0,Y 523.968,Z 580.211,A -85,B 0,C 180,E1 -4845.235,E2 -4845.235} C_VEL
LIN {X 0,Y 524.007,Z 580.216,A -85,B 0,C 180,E1 -4848.394,E2 -4848.394} C_VEL
LIN {X 0,Y 524,Z 580.209,A -85,B 0,C 180,E1 -4851.516,E2 -4851.516} C_VEL
LIN {X 0,Y 524.077,Z 580.204,A -85,B 0,C 180,E1 -4854.614,E2 -4854.614} C_VEL
LIN {X 0,Y 524.104,Z 580.197,A -85,B 0,C 180,E1 -4857.694,E2 -4857.694} C_VEL
LIN {X 0,Y 524.117,Z 580.197,A -85,B 0,C 180,E1 -4860.768,E2 -4860.768} C_VEL
LIN {X 0,Y 524.068,Z 580.201,A -85,B 0,C 180,E1 -4863.075,E2 -4863.075} C_VEL
LIN {X 0,Y 524.045,Z 580.212,A -85,B 0,C 180,E1 -4866.159,E2 -4866.159} C_VEL
LIN {X 0,Y 523.997,Z 580.21,A -85,B 0,C 180,E1 -4869.262,E2 -4869.262} C_VEL
LIN {X 0,Y 524.016,Z 580.209,A -85,B 0,C 180,E1 -4871.751,E2 -4871.751} C_VEL
LIN {X 0,Y 523.968,Z 580.219,A -85,B 0,C 180,E1 -4875.046,E2 -4875.046} C_VEL
LIN {X 0,Y 524.038,Z 580.418,A -85,B 0,C 180,E1 -4876.809,E2 -4876.809} C_VEL
LIN {X 0,Y 524.342,Z 585.631,A -85,B 0,C 180,E1 -4877.955,E2 -4877.955} C_VEL
LIN {X 0,Y 524.048,Z 594.617,A -85,B 0,C 180,E1 -4879.903,E2 -4879.903} C_VEL
LIN {X 0,Y 525.918,Z 604.354,A -85,B 0,C 180,E1 -4880.106,E2 -4880.106} C_VEL
LIN {X 0,Y 525.507,Z 700.625,A -85,B 0,C 180,E1 -4881.45,E2 -4881.45} C_VEL
LIN {X 0,Y 525.3,Z 713.065,A -85,B 0,C 180,E1 -4881.768,E2 -4881.768} C_VEL
LIN {X 0,Y 525.106,Z 725.449,A -85,B 0,C 180,E1 -4882.231,E2 -4882.231} C_VEL
LIN {X 0,Y 524.85,Z 737.491,A -85,B 0,C 180,E1 -4882.85,E2 -4882.85} C_VEL
LIN {X 0,Y 524.574,Z 748.687,A -85,B 0,C 180,E1 -4883.594,E2 -4883.594} C_VEL
LIN {X 0,Y 524.289,Z 758.256,A -85,B 0,C 180,E1 -4884.381,E2 -4884.381} C_VEL
LIN {X 0,Y 524.055,Z 767.065,A -85,B 0,C 180,E1 -4885.267,E2 -4885.267} C_VEL
LIN {X 0,Y 523.78,Z 775.386,A -85,B 0,C 180,E1 -4886.282,E2 -4886.282} C_VEL
